LIN {X 0,Y 474.608,Z 876.179,A -85,B 0,C 180,E1 -7254.724,E2 -7254.724} C_VEL
LIN {X 0,Y 474.616,Z 876.172,A -85,B 0,C 180,E1 -7257.786,E2 -7257.786} C_VEL
LIN {X 0,Y 474.574,Z 876.184,A -85,B 0,C 180,E1 -7260.895,E2 -7260.895} C_VEL
LIN {X 0,Y 474.57,Z 876.184,A -85,B 0,C 180,E1 -7263.623,E2 -7263.623} C_VEL
LIN {X 0,Y 474.646,Z 876.303,A -85,B 0,C 180,E1 -7265.768,E2 -7265.768} C_VEL
LIN {X 0,Y 476.171,Z 885.136,A -85,B 0,C 180,E1 -7267.663,E2 -7267.663} C_VEL
LIN {X 0,Y 475.761,Z 898.657,A -85,B 0,C 180,E1 -7270.362,E2 -7270.362} C_VEL
LIN {X 0,Y 475.106,Z 915.52,A -85,B 0,C 180,E1 -7273.676,E2 -7273.676} C_VEL
LIN {X 0,Y 474.617,Z 931.729,A -85,B 0,C 180,E1 -7276.845,E2 -7276.845} C_VEL
LIN {X 0,Y 476.334,Z 945.669,A -85,B 0,C 180,E1 -7277.131,E2 -7277.131} C_VEL
LIN {X 0,Y 476.068,Z 1005.948,A -85,B 0,C 180,E1 -7278.072,E2 -7278.072} C_VEL
LIN {X 0,Y 475.814,Z 1016.704,A -85,B 0,C 180,E1 -7278.336,E2 -7278.336} C_VEL
LIN {X 0,Y 475.639,Z 1025.306,A -85,B 0,C 180,E1 -7278.656,E2 -7278.656} C_VEL
LIN {X 0,Y 475.412,Z 1032.974,A -85,B 0,C 180,E1 -7279.028,E2 -7279.028} C_VEL
LIN {X 0,Y 475.18,Z 1041.593,A -85,B 0,C 180,E1 -7279.561,E2 -7279.561} C_VEL
LIN {X 0,Y 474.915,Z 1049.857,A -85,B 0,C 180,E1 -7280.201,E2 -7280.201} C_VEL
LIN {X 0,Y 474.663,Z 1057.701,A -85,B 0,C 180,E1 -7280.949,E2 -7280.949} C_VEL
LIN {X 0,Y 474.415,Z 1064.184,A -85,B 0,C 180,E1 -7281.695,E2 -7281.695} C_VEL
LIN {X 0,Y 474.228,Z 1070.364,A -85,B 0,C 180,E1 -7282.549,E2 -7282.549} C_VEL
LIN {X 0,Y 474.034,Z 1076.736,A -85,B 0,C 180,E1 -7283.626,E2 -7283.626} C_VEL
LIN {X 0,Y 473.878,Z 1082.509,A -85,B 0,C 180,E1 -7284.895,E2 -7284.895} C_VEL
LIN {X 0,Y 473.799,Z 1085.552,A -85,B 0,C 180,E1 -7285.746,E2 -7285.746} C_VEL
LIN {X 0,Y 473.852,Z 1087.914,A -85,B 0,C 180,E1 -7286.599,E2 -7286.599} C_VEL
LIN {X 0,Y 473.745,Z 1089.693,A -85,B 0,C 180,E1 -7287.449,E2 -7287.449} C_VEL
LIN {X 0,Y 473.723,Z 1090.971,A -85,B 0,C 180,E1 -7288.3,E2 -7288.3} C_VEL
LIN {X 0,Y 473.685,Z 1091.763,A -85,B 0,C 180,E1 -7289.15,E2 -7289.15} C_VEL
LIN {X 0,Y 473.666,Z 1092.054,A -85,B 0,C 180,E1 -7290,E2 -7290} C_VEL
LIN {X 0,Y 473.685,Z 1091.749,A -85,B 0,C 180,E1 -7290.85,E2 -7290.85} C_VEL
LIN {X 0,Y 473.723,Z 1090.953,A -85,B 0,C 180,E1 -7291.7,E2 -7291.7} C_VEL
LIN {X 0,Y 473.745,Z 1089.662,A -85,B 0,C 180,E1 -7292.551,E2 -7292.551} C_VEL
LIN {X 0,Y 473.852,Z 1086.693,A -85,B 0,C 180,E1 -7293.827,E2 -7293.827} C_VEL
LIN {X 0,Y 473.878,Z 1082.413,A -85,B 0,C 180,E1 -7295.105,E2 -7295.105} C_VEL
LIN {X 0,Y 474.038,Z 1076.567,A -85,B 0,C 180,E1 -7296.38,E2 -7296.38} C_VEL
LIN {X 0,Y 474.228,Z 1070.202,A -85,B 0,C 180,E1 -7297.451,E2 -7297.451} C_VEL
LIN {X 0,Y 474.391,Z 1063.985,A -85,B 0,C 180,E1 -7298.305,E2 -7298.305} C_VEL
LIN {X 0,Y 474.656,Z 1056.411,A -85,B 0,C 180,E1 -7299.159,E2 -7299.159} C_VEL
LIN {X 0,Y 474.931,Z 1048.281,A -85,B 0,C 180,E1 -7299.906,E2 -7299.906} C_VEL
LIN {X 0,Y 475.267,Z 1038.079,A -85,B 0,C 180,E1 -7300.652,E2 -7300.652} C_VEL
LIN {X 0,Y 475.519,Z 1027.086,A -85,B 0,C 180,E1 -7301.239,E2 -7301.239} C_VEL
LIN {X 0,Y 475.754,Z 1017.515,A -85,B 0,C 180,E1 -7301.611,E2 -7301.611} C_VEL
LIN {X 0,Y 475.986,Z 1008.593,A -85,B 0,C 180,E1 -7301.849,E2 -7301.849} C_VEL
LIN {X 0,Y 476.181,Z 944.23,A -85,B 0,C 180,E1 -7302.888,E2 -7302.888} C_VEL
LIN {X 0,Y 474.612,Z 931.089,A -85,B 0,C 180,E1 -7303.172,E2 -7303.172} C_VEL
LIN {X 0,Y 475.08,Z 913.604,A -85,B 0,C 180,E1 -7306.545,E2 -7306.545} C_VEL
LIN {X 0,Y 475.627,Z 897.776,A -85,B 0,C 180,E1 -7309.643,E2 -7309.643} C_VEL
LIN {X 0,Y 476.054,Z 884.31,A -85,B 0,C 180,E1 -7312.343,E2 -7312.343} C_VEL
LIN {X 0,Y 474.644,Z 876.176,A -85,B 0,C 180,E1 -7314.144,E2 -7314.144} C_VEL
LIN {X 0,Y 474.59,Z 876.184,A -85,B 0,C 180,E1 -7317.327,E2 -7317.327} C_VEL
LIN {X 0,Y 474.547,Z 876.183,A -85,B 0,C 180,E1 -7320.234,E2 -7320.234} C_VEL
LIN {X 0,Y 474.61,Z 876.182,A -85,B 0,C 180,E1 -7323.223,E2 -7323.223} C_VEL
LIN {X 0,Y 474.564,Z 876.18,A -85,B 0,C 180,E1 -7326.326,E2 -7326.326} C_VEL
LIN {X 0,Y 474.594,Z 876.182,A -85,B 0,C 180,E1 -7329.551,E2 -7329.551} C_VEL
LIN {X 0,Y 474.562,Z 876.181,A -85,B 0,C 180,E1 -7332.94,E2 -7332.94} C_VEL
LIN {X 0,Y 474.595,Z 876.182,A -85,B 0,C 180,E1 -7335.894,E2 -7335.894} C_VEL
LIN {X 0,Y 474.578,Z 876.178,A -85,B 0,C 180,E1 -7339.048,E2 -7339.048} C_VEL
LIN {X 0,Y 474.58,Z 876.181,A -85,B 0,C 180,E1 -7341.709,E2 -7341.709} C_VEL
LIN {X 0,Y 474.607,Z 876.178,A -85,B 0,C 180,E1 -7344.724,E2 -7344.724} C_VEL
LIN {X 0,Y 474.615,Z 876.175,A -85,B 0,C 180,E1 -7347.786,E2 -7347.786} C_VEL
LIN {X 0,Y 474.573,Z 876.185,A -85,B 0,C 180,E1 -7350.896,E2 -7350.896} C_VEL
LIN {X 0,Y 474.569,Z 876.181,A -85,B 0,C 180,E1 -7353.623,E2 -7353.623} C_VEL
LIN {X 0,Y 474.594,Z 876.185,A -85,B 0,C 180,E1 -7356.653,E2 -7356.653} C_VEL
LIN {X 0,Y 474.647,Z 876.177,A -85,B 0,C 180,E1 -7359.185,E2 -7359.185} C_VEL
LIN {X 0,Y 474.67,Z 876.361,A -85,B 0,C 180,E1 -7361.496,E2 -7361.496} C_VEL
LIN {X 0,Y 475.011,Z 881.021,A -85,B 0,C 180,E1 -7362.788,E2 -7362.788} C_VEL
LIN {X 0,Y 474.637,Z 892.536,A -85,B 0,C 180,E1 -7365.859,E2 -7365.859} C_VEL
LIN {X 0,Y 474.532,Z 896.576,A -85,B 0,C 180,E1 -7366.925,E2 -7366.925} C_VEL
LIN {X 0,Y 476.468,Z 909.333,A -85,B 0,C 180,E1 -7367.193,E2 -7367.193} C_VEL
LIN {X 0,Y 475.939,Z 972.842,A -85,B 0,C 180,E1 -7368.232,E2 -7368.232} C_VEL
LIN {X 0,Y 475.768,Z 983.733,A -85,B 0,C 180,E1 -7368.551,E2 -7368.551} C_VEL
LIN {X 0,Y 475.515,Z 994.365,A -85,B 0,C 180,E1 -7369.031,E2 -7369.031} C_VEL
LIN {X 0,Y 475.301,Z 1003.198,A -85,B 0,C 180,E1 -7369.565,E2 -7369.565} C_VEL
LIN {X 0,Y 475.061,Z 1011.606,A -85,B 0,C 180,E1 -7370.205,E2 -7370.205} C_VEL
LIN {X 0,Y 474.793,Z 1019.544,A -85,B 0,C 180,E1 -7370.952,E2 -7370.952} C_VEL
LIN {X 0,Y 474.52,Z 1026.089,A -85,B 0,C 180,E1 -7371.698,E2 -7371.698} C_VEL
LIN {X 0,Y 474.314,Z 1032.298,A -85,B 0,C 180,E1 -7372.551,E2 -7372.551} C_VEL
LIN {X 0,Y 474.173,Z 1038.052,A -85,B 0,C 180,E1 -7373.515,E2 -7373.515} C_VEL
LIN {X 0,Y 474.005,Z 1042.684,A -85,B 0,C 180,E1 -7374.47,E2 -7374.47} C_VEL
LIN {X 0,Y 473.892,Z 1046.03,A -85,B 0,C 180,E1 -7375.322,E2 -7375.322} C_VEL
LIN {X 0,Y 473.894,Z 1048.738,A -85,B 0,C 180,E1 -7376.174,E2 -7376.174} C_VEL
LIN {X 0,Y 473.756,Z 1051.695,A -85,B 0,C 180,E1 -7377.45,E2 -7377.45} C_VEL
LIN {X 0,Y 473.753,Z 1052.994,A -85,B 0,C 180,E1 -7378.3,E2 -7378.3} C_VEL
LIN {X 0,Y 473.686,Z 1053.81,A -85,B 0,C 180,E1 -7379.15,E2 -7379.15} C_VEL
LIN {X 0,Y 473.667,Z 1054.103,A -85,B 0,C 180,E1 -7380,E2 -7380} C_VEL
LIN {X 0,Y 473.686,Z 1053.826,A -85,B 0,C 180,E1 -7380.851,E2 -7380.851} C_VEL
LIN {X 0,Y 473.753,Z 1053.066,A -85,B 0,C 180,E1 -7381.701,E2 -7381.701} C_VEL
LIN {X 0,Y 473.746,Z 1051.823,A -85,B 0,C 180,E1 -7382.551,E2 -7382.551} C_VEL
LIN {X 0,Y 473.889,Z 1048.918,A -85,B 0,C 180,E1 -7383.827,E2 -7383.827} C_VEL
LIN {X 0,Y 473.878,Z 1044.748,A -85,B 0,C 180,E1 -7385.106,E2 -7385.106} C_VEL
LIN {X 0,Y 474.197,Z 1039.865,A -85,B 0,C 180,E1 -7386.22,E2 -7386.22} C_VEL
LIN {X 0,Y 474.292,Z 1032.814,A -85,B 0,C 180,E1 -7387.45,E2 -7387.45} C_VEL
LIN {X 0,Y 474.473,Z 1026.718,A -85,B 0,C 180,E1 -7388.304,E2 -7388.304} C_VEL
LIN {X 0,Y 474.766,Z 1019.299,A -85,B 0,C 180,E1 -7389.157,E2 -7389.157} C_VEL
LIN {X 0,Y 475.078,Z 1011.356,A -85,B 0,C 180,E1 -7389.903,E2 -7389.903} C_VEL
LIN {X 0,Y 475.355,Z 1001.42,A -85,B 0,C 180,E1 -7390.65,E2 -7390.65} C_VEL
LIN {X 0,Y 475.61,Z 990.9,A -85,B 0,C 180,E1 -7391.238,E2 -7391.238} C_VEL
LIN {X 0,Y 475.793,Z 981.013,A -85,B 0,C 180,E1 -7391.638,E2 -7391.638} C_VEL
LIN {X 0,Y 476.004,Z 971.331,A -85,B 0,C 180,E1 -7391.903,E2 -7391.903} C_VEL
LIN {X 0,Y 476.316,Z 907.193,A -85,B 0,C 180,E1 -7392.941,E2 -7392.941} C_VEL
LIN {X 0,Y 474.447,Z 895.857,A -85,B 0,C 180,E1 -7393.198,E2 -7393.198} C_VEL
LIN {X 0,Y 474.781,Z 883.788,A -85,B 0,C 180,E1 -7396.335,E2 -7396.335} C_VEL
LIN {X 0,Y 474.736,Z 876.329,A -85,B 0,C 180,E1 -7398.305,E2 -7398.305} C_VEL
LIN {X 0,Y 474.579,Z 876.178,A -85,B 0,C 180,E1 -7401.73,E2 -7401.73} C_VEL
LIN {X 0,Y 474.586,Z 876.177,A -85,B 0,C 180,E1 -7404.497,E2 -7404.497} C_VEL
LIN {X 0,Y 474.594,Z 876.184,A -85,B 0,C 180,E1 -7407.327,E2 -7407.327} C_VEL
LIN {X 0,Y 474.551,Z 876.181,A -85,B 0,C 180,E1 -7410.235,E2 -7410.235} C_VEL
LIN {X 0,Y 474.614,Z 876.176,A -85,B 0,C 180,E1 -7413.223,E2 -7413.223} C_VEL
LIN {X 0,Y 474.571,Z 876.18,A -85,B 0,C 180,E1 -7416.326,E2 -7416.326} C_VEL
LIN {X 0,Y 474.6,Z 876.178,A -85,B 0,C 180,E1 -7419.551,E2 -7419.551} C_VEL
LIN {X 0,Y 474.568,Z 876.178,A -85,B 0,C 180,E1 -7422.94,E2 -7422.94} C_VEL
LIN {X 0,Y 474.6,Z 876.179,A -85,B 0,C 180,E1 -7425.894,E2 -7425.894} C_VEL
LIN {X 0,Y 474.582,Z 876.177,A -85,B 0,C 180,E1 -7429.048,E2 -7429.048} C_VEL
LIN {X 0,Y 474.586,Z 876.177,A -85,B 0,C 180,E1 -7431.709,E2 -7431.709} C_VEL
LIN {X 0,Y 474.613,Z 876.179,A -85,B 0,C 180,E1 -7434.725,E2 -7434.725} C_VEL
LIN {X 0,Y 474.62,Z 876.172,A -85,B 0,C 180,E1 -7437.787,E2 -7437.787} C_VEL
LIN {X 0,Y 474.574,Z 876.183,A -85,B 0,C 180,E1 -7441.04,E2 -7441.04} C_VEL
LIN {X 0,Y 473.906,Z 876.263,A -85,B 0,C 180,E1 -7441.749,E2 -7441.749} C_VEL
LIN {X 0,Y 471.064,Z 876.624,A -85,B 0,C 180,E1 -7442.899,E2 -7442.899} C_VEL
LIN {X 0,Y 468.663,Z 876.918,A -85,B 0,C 180,E1 -7443.826,E2 -7443.826} C_VEL
LIN {X 0,Y 467.633,Z 877.045,A -85,B 0,C 180,E1 -7444.542,E2 -7444.542} C_VEL
LIN {X 0,Y 467.55,Z 877.056,A -85,B 0,C 180,E1 -7444.785,E2 -7444.785} C_VEL
LIN {X 0,Y 467.555,Z 877.059,A -85,B 0,C 180,E1 -7446.995,E2 -7446.995} C_VEL
LIN {X 0,Y 467.597,Z 877.049,A -85,B 0,C 180,E1 -7449.776,E2 -7449.776} C_VEL
LIN {X 0,Y 467.58,Z 877.049,A -85,B 0,C 180,E1 -7452.506,E2 -7452.506} C_VEL
LIN {X 0,Y 467.599,Z 877.051,A -85,B 0,C 180,E1 -7455.196,E2 -7455.196} C_VEL
LIN {X 0,Y 467.64,Z 877.046,A -85,B 0,C 180,E1 -7457.854,E2 -7457.854} C_VEL
LIN {X 0,Y 467.633,Z 877.046,A -85,B 0,C 180,E1 -7461.356,E2 -7461.356} C_VEL
LIN {X 0,Y 467.704,Z 877.04,A -85,B 0,C 180,E1 -7463.962,E2 -7463.962} C_VEL
LIN {X 0,Y 467.786,Z 877.025,A -85,B 0,C 180,E1 -7467.417,E2 -7467.417} C_VEL
LIN {X 0,Y 467.852,Z 877.022,A -85,B 0,C 180,E1 -7470,E2 -7470} C_VEL
LIN {X 0,Y 467.784,Z 877.027,A -85,B 0,C 180,E1 -7472.583,E2 -7472.583} C_VEL
LIN {X 0,Y 467.704,Z 877.037,A -85,B 0,C 180,E1 -7476.038,E2 -7476.038} C_VEL
LIN {X 0,Y 467.633,Z 877.048,A -85,B 0,C 180,E1 -7478.644,E2 -7478.644} C_VEL
LIN {X 0,Y 467.644,Z 877.045,A -85,B 0,C 180,E1 -7482.348,E2 -7482.348} C_VEL
LIN {X 0,Y 467.578,Z 877.049,A -85,B 0,C 180,E1 -7485.852,E2 -7485.852} C_VEL
LIN {X 0,Y 467.578,Z 877.055,A -85,B 0,C 180,E1 -7488.748,E2 -7488.748} C_VEL
LIN {X 0,Y 467.571,Z 877.055,A -85,B 0,C 180,E1 -7491.263,E2 -7491.263} C_VEL
LIN {X 0,Y 467.536,Z 877.055,A -85,B 0,C 180,E1 -7493.946,E2 -7493.946} C_VEL
LIN {X 0,Y 467.529,Z 877.057,A -85,B 0,C 180,E1 -7496.806,E2 -7496.806} C_VEL
LIN {X 0,Y 467.514,Z 877.061,A -85,B 0,C 180,E1 -7499.741,E2 -7499.741} C_VEL
LIN {X 0,Y 467.549,Z 877.053,A -85,B 0,C 180,E1 -7502.761,E2 -7502.761} C_VEL
LIN {X 0,Y 467.542,Z 877.059,A -85,B 0,C 180,E1 -7505.891,E2 -7505.891} C_VEL
LIN {X 0,Y 467.53,Z 877.056,A -85,B 0,C 180,E1 -7509.15,E2 -7509.15} C_VEL
LIN {X 0,Y 467.553,Z 877.054,A -85,B 0,C 180,E1 -7511.406,E2 -7511.406} C_VEL
LIN {X 0,Y 467.566,Z 877.051,A -85,B 0,C 180,E1 -7515.052,E2 -7515.052} C_VEL
LIN {X 0,Y 467.553,Z 877.055,A -85,B 0,C 180,E1 -7518.727,E2 -7518.727} C_VEL
LIN {X 0,Y 467.536,Z 877.057,A -85,B 0,C 180,E1 -7521.952,E2 -7521.952} C_VEL
LIN {X 0,Y 467.553,Z 877.054,A -85,B 0,C 180,E1 -7525.166,E2 -7525.166} C_VEL
LIN {X 0,Y 467.55,Z 877.055,A -85,B 0,C 180,E1 -7528.257,E2 -7528.257} C_VEL
LIN {X 0,Y 467.528,Z 877.058,A -85,B 0,C 180,E1 -7531.247,E2 -7531.247} C_VEL
LIN {X 0,Y 467.565,Z 877.052,A -85,B 0,C 180,E1 -7534.405,E2 -7534.405} C_VEL
LIN {X 0,Y 467.555,Z 877.059,A -85,B 0,C 180,E1 -7536.994,E2 -7536.994} C_VEL
LIN {X 0,Y 467.596,Z 877.048,A -85,B 0,C 180,E1 -7539.775,E2 -7539.775} C_VEL
LIN {X 0,Y 467.579,Z 877.049,A -85,B 0,C 180,E1 -7542.505,E2 -7542.505} C_VEL
LIN {X 0,Y 467.571,Z 877.055,A -85,B 0,C 180,E1 -7545.195,E2 -7545.195} C_VEL
LIN {X 0,Y 467.638,Z 877.046,A -85,B 0,C 180,E1 -7547.854,E2 -7547.854} C_VEL
LIN {X 0,Y 467.631,Z 877.046,A -85,B 0,C 180,E1 -7551.356,E2 -7551.356} C_VEL
LIN {X 0,Y 467.702,Z 877.04,A -85,B 0,C 180,E1 -7553.962,E2 -7553.962} C_VEL
LIN {X 0,Y 467.783,Z 877.025,A -85,B 0,C 180,E1 -7557.416,E2 -7557.416} C_VEL
LIN {X 0,Y 467.85,Z 877.022,A -85,B 0,C 180,E1 -7560,E2 -7560} C_VEL
LIN {X 0,Y 467.782,Z 877.027,A -85,B 0,C 180,E1 -7562.583,E2 -7562.583} C_VEL
LIN {X 0,Y 467.701,Z 877.038,A -85,B 0,C 180,E1 -7566.038,E2 -7566.038} C_VEL
LIN {X 0,Y 467.63,Z 877.048,A -85,B 0,C 180,E1 -7568.643,E2 -7568.643} C_VEL
LIN {X 0,Y 467.64,Z 877.046,A -85,B 0,C 180,E1 -7572.348,E2 -7572.348} C_VEL
LIN {X 0,Y 467.575,Z 877.049,A -85,B 0,C 180,E1 -7575.851,E2 -7575.851} C_VEL
LIN {X 0,Y 467.574,Z 877.055,A -85,B 0,C 180,E1 -7578.747,E2 -7578.747} C_VEL
LIN {X 0,Y 467.568,Z 877.055,A -85,B 0,C 180,E1 -7581.263,E2 -7581.263} C_VEL
LIN {X 0,Y 467.532,Z 877.055,A -85,B 0,C 180,E1 -7583.945,E2 -7583.945} C_VEL
LIN {X 0,Y 467.525,Z 877.058,A -85,B 0,C 180,E1 -7586.806,E2 -7586.806} C_VEL
LIN {X 0,Y 467.51,Z 877.061,A -85,B 0,C 180,E1 -7589.741,E2 -7589.741} C_VEL
LIN {X 0,Y 467.545,Z 877.053,A -85,B 0,C 180,E1 -7592.761,E2 -7592.761} C_VEL
LIN {X 0,Y 467.538,Z 877.059,A -85,B 0,C 180,E1 -7595.891,E2 -7595.891} C_VEL
LIN {X 0,Y 467.526,Z 877.056,A -85,B 0,C 180,E1 -7599.15,E2 -7599.15} C_VEL
LIN {X 0,Y 467.549,Z 877.054,A -85,B 0,C 180,E1 -7601.406,E2 -7601.406} C_VEL
LIN {X 0,Y 467.561,Z 877.051,A -85,B 0,C 180,E1 -7605.051,E2 -7605.051} C_VEL
LIN {X 0,Y 467.549,Z 877.055,A -85,B 0,C 180,E1 -7608.727,E2 -7608.727} C_VEL
LIN {X 0,Y 467.532,Z 877.057,A -85,B 0,C 180,E1 -7611.952,E2 -7611.952} C_VEL
LIN {X 0,Y 467.548,Z 877.054,A -85,B 0,C 180,E1 -7615.166,E2 -7615.166} C_VEL
LIN {X 0,Y 467.545,Z 877.056,A -85,B 0,C 180,E1 -7618.257,E2 -7618.257} C_VEL
LIN {X 0,Y 467.523,Z 877.058,A -85,B 0,C 180,E1 -7621.247,E2 -7621.247} C_VEL
LIN {X 0,Y 467.56,Z 877.059,A -85,B 0,C 180,E1 -7624.405,E2 -7624.405} C_VEL
LIN {X 0,Y 467.611,Z 877.113,A -85,B 0,C 180,E1 -7625.587,E2 -7625.587} C_VEL
LIN {X 0,Y 469.195,Z 886.106,A -85,B 0,C 180,E1 -7627.545,E2 -7627.545} C_VEL
LIN {X 0,Y 468.755,Z 899.583,A -85,B 0,C 180,E1 -7630.285,E2 -7630.285} C_VEL
LIN {X 0,Y 468.122,Z 915.269,A -85,B 0,C 180,E1 -7633.426,E2 -7633.426} C_VEL
LIN {X 0,Y 467.562,Z 931.496,A -85,B 0,C 180,E1 -7636.646,E2 -7636.646} C_VEL
LIN {X 0,Y 469.42,Z 946.323,A -85,B 0,C 180,E1 -7636.955,E2 -7636.955} C_VEL
LIN {X 0,Y 469.069,Z 1007.527,A -85,B 0,C 180,E1 -7637.946,E2 -7637.946} C_VEL
LIN {X 0,Y 468.81,Z 1017.577,A -85,B 0,C 180,E1 -7638.214,E2 -7638.214} C_VEL
LIN {X 0,Y 468.597,Z 1027.069,A -85,B 0,C 180,E1 -7638.592,E2 -7638.592} C_VEL
LIN {X 0,Y 468.297,Z 1038,A -85,B 0,C 180,E1 -7639.187,E2 -7639.187} C_VEL
LIN {X 0,Y 467.948,Z 1048.161,A -85,B 0,C 180,E1 -7639.945,E2 -7639.945} C_VEL
LIN {X 0,Y 467.617,Z 1056.243,A -85,B 0,C 180,E1 -7640.702,E2 -7640.702} C_VEL
LIN {X 0,Y 467.424,Z 1062.068,A -85,B 0,C 180,E1 -7641.352,E2 -7641.352} C_VEL
LIN {X 0,Y 467.182,Z 1068.557,A -85,B 0,C 180,E1 -7642.219,E2 -7642.219} C_VEL
LIN {X 0,Y 467.042,Z 1073.953,A -85,B 0,C 180,E1 -7643.086,E2 -7643.086} C_VEL
LIN {X 0,Y 466.926,Z 1078.452,A -85,B 0,C 180,E1 -7643.952,E2 -7643.952} C_VEL
LIN {X 0,Y 466.815,Z 1082.195,A -85,B 0,C 180,E1 -7644.817,E2 -7644.817} C_VEL
LIN {X 0,Y 466.707,Z 1085.246,A -85,B 0,C 180,E1 -7645.682,E2 -7645.682} C_VEL
LIN {X 0,Y 466.766,Z 1087.616,A -85,B 0,C 180,E1 -7646.547,E2 -7646.547} C_VEL
LIN {X 0,Y 466.668,Z 1089.404,A -85,B 0,C 180,E1 -7647.41,E2 -7647.41} C_VEL
LIN {X 0,Y 466.63,Z 1090.686,A -85,B 0,C 180,E1 -7648.274,E2 -7648.274} C_VEL
LIN {X 0,Y 466.616,Z 1091.482,A -85,B 0,C 180,E1 -7649.137,E2 -7649.137} C_VEL
LIN {X 0,Y 466.595,Z 1091.772,A -85,B 0,C 180,E1 -7650,E2 -7650} C_VEL
LIN {X 0,Y 466.616,Z 1091.463,A -85,B 0,C 180,E1 -7650.863,E2 -7650.863} C_VEL
LIN {X 0,Y 466.63,Z 1090.657,A -85,B 0,C 180,E1 -7651.726,E2 -7651.726} C_VEL
LIN {X 0,Y 466.667,Z 1089.362,A -85,B 0,C 180,E1 -7652.589,E2 -7652.589} C_VEL
LIN {X 0,Y 466.744,Z 1086.368,A -85,B 0,C 180,E1 -7653.885,E2 -7653.885} C_VEL
LIN {X 0,Y 466.815,Z 1082.069,A -85,B 0,C 180,E1 -7655.183,E2 -7655.183} C_VEL
LIN {X 0,Y 466.94,Z 1076.869,A -85,B 0,C 180,E1 -7656.35,E2 -7656.35} C_VEL
LIN {X 0,Y 467.16,Z 1069.782,A -85,B 0,C 180,E1 -7657.564,E2 -7657.564} C_VEL
LIN {X 0,Y 467.349,Z 1063.524,A -85,B 0,C 180,E1 -7658.431,E2 -7658.431} C_VEL
LIN {X 0,Y 467.593,Z 1056.95,A -85,B 0,C 180,E1 -7659.189,E2 -7659.189} C_VEL
LIN {X 0,Y 467.862,Z 1048.981,A -85,B 0,C 180,E1 -7659.947,E2 -7659.947} C_VEL
LIN {X 0,Y 468.195,Z 1040.575,A -85,B 0,C 180,E1 -7660.596,E2 -7660.596} C_VEL
LIN {X 0,Y 468.44,Z 1029.847,A -85,B 0,C 180,E1 -7661.247,E2 -7661.247} C_VEL
LIN {X 0,Y 468.716,Z 1019.047,A -85,B 0,C 180,E1 -7661.706,E2 -7661.706} C_VEL
LIN {X 0,Y 469,Z 1008.617,A -85,B 0,C 180,E1 -7662,E2 -7662} C_VEL
LIN {X 0,Y 469.312,Z 945.308,A -85,B 0,C 180,E1 -7663.056,E2 -7663.056} C_VEL
LIN {X 0,Y 467.557,Z 930.956,A -85,B 0,C 180,E1 -7663.351,E2 -7663.351} C_VEL
LIN {X 0,Y 467.945,Z 916.235,A -85,B 0,C 180,E1 -7666.222,E2 -7666.222} C_VEL
LIN {X 0,Y 468.572,Z 899.794,A -85,B 0,C 180,E1 -7669.495,E2 -7669.495} C_VEL
LIN {X 0,Y 469.119,Z 886.391,A -85,B 0,C 180,E1 -7672.227,E2 -7672.227} C_VEL
LIN {X 0,Y 467.586,Z 877.056,A -85,B 0,C 180,E1 -7674.296,E2 -7674.296} C_VEL
LIN {X 0,Y 467.535,Z 877.06,A -85,B 0,C 180,E1 -7677.774,E2 -7677.774} C_VEL
LIN {X 0,Y 467.525,Z 877.064,A -85,B 0,C 180,E1 -7681.036,E2 -7681.036} C_VEL
LIN {X 0,Y 467.564,Z 877.057,A -85,B 0,C 180,E1 -7683.79,E2 -7683.79} C_VEL
LIN {X 0,Y 467.496,Z 877.062,A -85,B 0,C 180,E1 -7686.965,E2 -7686.965} C_VEL
LIN {X 0,Y 467.519,Z 877.062,A -85,B 0,C 180,E1 -7689.946,E2 -7689.946} C_VEL
LIN {X 0,Y 467.514,Z 877.059,A -85,B 0,C 180,E1 -7692.569,E2 -7692.569} C_VEL
LIN {X 0,Y 467.559,Z 877.053,A -85,B 0,C 180,E1 -7695.052,E2 -7695.052} C_VEL
LIN {X 0,Y 467.547,Z 877.055,A -85,B 0,C 180,E1 -7698.728,E2 -7698.728} C_VEL
LIN {X 0,Y 467.531,Z 877.062,A -85,B 0,C 180,E1 -7701.953,E2 -7701.953} C_VEL
LIN {X 0,Y 467.547,Z 877.054,A -85,B 0,C 180,E1 -7705.166,E2 -7705.166} C_VEL
LIN {X 0,Y 467.544,Z 877.06,A -85,B 0,C 180,E1 -7708.257,E2 -7708.257} C_VEL
LIN {X 0,Y 467.522,Z 877.059,A -85,B 0,C 180,E1 -7711.247,E2 -7711.247} C_VEL
LIN {X 0,Y 467.559,Z 877.058,A -85,B 0,C 180,E1 -7714.406,E2 -7714.406} C_VEL
LIN {X 0,Y 467.545,Z 877.064,A -85,B 0,C 180,E1 -7716.995,E2 -7716.995} C_VEL
LIN {X 0,Y 467.591,Z 877.053,A -85,B 0,C 180,E1 -7719.776,E2 -7719.776} C_VEL
LIN {X 0,Y 467.588,Z 877.123,A -85,B 0,C 180,E1 -7721.305,E2 -7721.305} C_VEL
LIN {X 0,Y 468.029,Z 881.408,A -85,B 0,C 180,E1 -7722.523,E2 -7722.523} C_VEL
LIN {X 0,Y 467.672,Z 891.243,A -85,B 0,C 180,E1 -7725.199,E2 -7725.199} C_VEL
LIN {X 0,Y 467.527,Z 896.94,A -85,B 0,C 180,E1 -7726.726,E2 -7726.726} C_VEL
LIN {X 0,Y 469.535,Z 909.305,A -85,B 0,C 180,E1 -7727.001,E2 -7727.001} C_VEL
LIN {X 0,Y 468.987,Z 972.192,A -85,B 0,C 180,E1 -7728.055,E2 -7728.055} C_VEL
LIN {X 0,Y 468.812,Z 982.59,A -85,B 0,C 180,E1 -7728.352,E2 -7728.352} C_VEL
LIN {X 0,Y 468.527,Z 994.306,A -85,B 0,C 180,E1 -7728.865,E2 -7728.865} C_VEL
LIN {X 0,Y 468.266,Z 1004.715,A -85,B 0,C 180,E1 -7729.515,E2 -7729.515} C_VEL
LIN {X 0,Y 468.012,Z 1012.911,A -85,B 0,C 180,E1 -7730.165,E2 -7730.165} C_VEL
LIN {X 0,Y 467.729,Z 1020.686,A -85,B 0,C 180,E1 -7730.923,E2 -7730.923} C_VEL
LIN {X 0,Y 467.38,Z 1029.614,A -85,B 0,C 180,E1 -7732.005,E2 -7732.005} C_VEL
LIN {X 0,Y 467.152,Z 1036.985,A -85,B 0,C 180,E1 -7733.182,E2 -7733.182} C_VEL
LIN {X 0,Y 467.103,Z 1040.992,A -85,B 0,C 180,E1 -7733.955,E2 -7733.955} C_VEL
LIN {X 0,Y 466.826,Z 1044.754,A -85,B 0,C 180,E1 -7734.818,E2 -7734.818} C_VEL
LIN {X 0,Y 466.829,Z 1048.999,A -85,B 0,C 180,E1 -7736.116,E2 -7736.116} C_VEL
LIN {X 0,Y 466.677,Z 1051.965,A -85,B 0,C 180,E1 -7737.411,E2 -7737.411} C_VEL
LIN {X 0,Y 466.672,Z 1053.267,A -85,B 0,C 180,E1 -7738.274,E2 -7738.274} C_VEL
LIN {X 0,Y 466.617,Z 1054.087,A -85,B 0,C 180,E1 -7739.137,E2 -7739.137} C_VEL
LIN {X 0,Y 466.596,Z 1054.387,A -85,B 0,C 180,E1 -7740,E2 -7740} C_VEL
LIN {X 0,Y 466.618,Z 1054.098,A -85,B 0,C 180,E1 -7740.863,E2 -7740.863} C_VEL
LIN {X 0,Y 466.658,Z 1053.328,A -85,B 0,C 180,E1 -7741.726,E2 -7741.726} C_VEL
LIN {X 0,Y 466.668,Z 1052.079,A -85,B 0,C 180,E1 -7742.59,E2 -7742.59} C_VEL
LIN {X 0,Y 466.821,Z 1049.157,A -85,B 0,C 180,E1 -7743.885,E2 -7743.885} C_VEL
LIN {X 0,Y 466.77,Z 1046.499,A -85,B 0,C 180,E1 -7744.751,E2 -7744.751} C_VEL
LIN {X 0,Y 467.104,Z 1041.28,A -85,B 0,C 180,E1 -7746.046,E2 -7746.046} C_VEL
LIN {X 0,Y 467.187,Z 1034.39,A -85,B 0,C 180,E1 -7747.347,E2 -7747.347} C_VEL
LIN {X 0,Y 467.45,Z 1026.839,A -85,B 0,C 180,E1 -7748.43,E2 -7748.43} C_VEL
LIN {X 0,Y 467.779,Z 1019.385,A -85,B 0,C 180,E1 -7749.295,E2 -7749.295} C_VEL
LIN {X 0,Y 468.079,Z 1011.397,A -85,B 0,C 180,E1 -7750.053,E2 -7750.053} C_VEL
LIN {X 0,Y 468.396,Z 1001.408,A -85,B 0,C 180,E1 -7750.811,E2 -7750.811} C_VEL
LIN {X 0,Y 468.651,Z 990.743,A -85,B 0,C 180,E1 -7751.407,E2 -7751.407} C_VEL
LIN {X 0,Y 468.825,Z 980.714,A -85,B 0,C 180,E1 -7751.813,E2 -7751.813} C_VEL
LIN {X 0,Y 469.032,Z 972.026,A -85,B 0,C 180,E1 -7752.055,E2 -7752.055} C_VEL
LIN {X 0,Y 469.337,Z 907.501,A -85,B 0,C 180,E1 -7753.133,E2 -7753.133} C_VEL
LIN {X 0,Y 467.443,Z 896.058,A -85,B 0,C 180,E1 -7753.404,E2 -7753.404} C_VEL
LIN {X 0,Y 467.755,Z 885.53,A -85,B 0,C 180,E1 -7756.174,E2 -7756.174} C_VEL
LIN {X 0,Y 467.835,Z 878.9,A -85,B 0,C 180,E1 -7757.937,E2 -7757.937} C_VEL
LIN {X 0,Y 467.66,Z 877.046,A -85,B 0,C 180,E1 -7758.459,E2 -7758.459} C_VEL
LIN {X 0,Y 467.568,Z 877.056,A -85,B 0,C 180,E1 -7761.264,E2 -7761.264} C_VEL
LIN {X 0,Y 467.534,Z 877.055,A -85,B 0,C 180,E1 -7763.946,E2 -7763.946} C_VEL
LIN {X 0,Y 467.526,Z 877.058,A -85,B 0,C 180,E1 -7766.806,E2 -7766.806} C_VEL
LIN {X 0,Y 467.511,Z 877.062,A -85,B 0,C 180,E1 -7769.742,E2 -7769.742} C_VEL
LIN {X 0,Y 467.573,Z 877.05,A -85,B 0,C 180,E1 -7772.76,E2 -7772.76} C_VEL
LIN {X 0,Y 467.544,Z 877.059,A -85,B 0,C 180,E1 -7775.891,E2 -7775.891} C_VEL
LIN {X 0,Y 467.53,Z 877.056,A -85,B 0,C 180,E1 -7779.151,E2 -7779.151} C_VEL
LIN {X 0,Y 467.551,Z 877.054,A -85,B 0,C 180,E1 -7781.406,E2 -7781.406} C_VEL
LIN {X 0,Y 467.564,Z 877.051,A -85,B 0,C 180,E1 -7785.052,E2 -7785.052} C_VEL
LIN {X 0,Y 467.552,Z 877.055,A -85,B 0,C 180,E1 -7788.728,E2 -7788.728} C_VEL
LIN {X 0,Y 467.538,Z 877.056,A -85,B 0,C 180,E1 -7791.953,E2 -7791.953} C_VEL
LIN {X 0,Y 467.552,Z 877.054,A -85,B 0,C 180,E1 -7795.166,E2 -7795.166} C_VEL
LIN {X 0,Y 467.549,Z 877.055,A -85,B 0,C 180,E1 -7798.257,E2 -7798.257} C_VEL
LIN {X 0,Y 467.528,Z 877.058,A -85,B 0,C 180,E1 -7801.247,E2 -7801.247} C_VEL
LIN {X 0,Y 467.565,Z 877.052,A -85,B 0,C 180,E1 -7804.406,E2 -7804.406} C_VEL
LIN {X 0,Y 467.55,Z 877.056,A -85,B 0,C 180,E1 -7804.785,E2 -7804.785} C_VEL
LIN {X 0,Y 466.89,Z 877.142,A -85,B 0,C 180,E1 -7805.503,E2 -7805.503} C_VEL
LIN {X 0,Y 464.06,Z 877.496,A -85,B 0,C 180,E1 -7806.671,E2 -7806.671} C_VEL
LIN {X 0,Y 461.657,Z 877.792,A -85,B 0,C 180,E1 -7807.612,E2 -7807.612} C_VEL
LIN {X 0,Y 460.613,Z 877.919,A -85,B 0,C 180,E1 -7808.339,E2 -7808.339} C_VEL
LIN {X 0,Y 460.521,Z 877.93,A -85,B 0,C 180,E1 -7808.585,E2 -7808.585} C_VEL
LIN {X 0,Y 460.535,Z 877.934,A -85,B 0,C 180,E1 -7811.309,E2 -7811.309} C_VEL
LIN {X 0,Y 460.591,Z 877.921,A -85,B 0,C 180,E1 -7814.059,E2 -7814.059} C_VEL
LIN {X 0,Y 460.606,Z 877.924,A -85,B 0,C 180,E1 -7817.666,E2 -7817.666} C_VEL
LIN {X 0,Y 460.588,Z 877.922,A -85,B 0,C 180,E1 -7821.223,E2 -7821.223} C_VEL
LIN {X 0,Y 460.67,Z 877.917,A -85,B 0,C 180,E1 -7823.87,E2 -7823.87} C_VEL
LIN {X 0,Y 460.733,Z 877.903,A -85,B 0,C 180,E1 -7827.377,E2 -7827.377} C_VEL
LIN {X 0,Y 460.822,Z 877.898,A -85,B 0,C 180,E1 -7830,E2 -7830} C_VEL
LIN {X 0,Y 460.731,Z 877.905,A -85,B 0,C 180,E1 -7832.623,E2 -7832.623} C_VEL
LIN {X 0,Y 460.671,Z 877.914,A -85,B 0,C 180,E1 -7836.131,E2 -7836.131} C_VEL
LIN {X 0,Y 460.588,Z 877.924,A -85,B 0,C 180,E1 -7838.777,E2 -7838.777} C_VEL
LIN {X 0,Y 460.602,Z 877.923,A -85,B 0,C 180,E1 -7842.435,E2 -7842.435} C_VEL
LIN {X 0,Y 460.531,Z 877.927,A -85,B 0,C 180,E1 -7845.965,E2 -7845.965} C_VEL
LIN {X 0,Y 460.536,Z 877.934,A -85,B 0,C 180,E1 -7848.887,E2 -7848.887} C_VEL
LIN {X 0,Y 460.516,Z 877.932,A -85,B 0,C 180,E1 -7851.486,E2 -7851.486} C_VEL
LIN {X 0,Y 460.498,Z 877.931,A -85,B 0,C 180,E1 -7854.335,E2 -7854.335} C_VEL
LIN {X 0,Y 460.489,Z 877.94,A -85,B 0,C 180,E1 -7857.249,E2 -7857.249} C_VEL
LIN {X 0,Y 460.482,Z 877.934,A -85,B 0,C 180,E1 -7860.242,E2 -7860.242} C_VEL
LIN {X 0,Y 460.502,Z 877.935,A -85,B 0,C 180,E1 -7863.327,E2 -7863.327} C_VEL
LIN {X 0,Y 460.458,Z 877.937,A -85,B 0,C 180,E1 -7866.531,E2 -7866.531} C_VEL
LIN {X 0,Y 460.495,Z 877.94,A -85,B 0,C 180,E1 -7869.867,E2 -7869.867} C_VEL
LIN {X 0,Y 460.46,Z 877.936,A -85,B 0,C 180,E1 -7872.892,E2 -7872.892} C_VEL
LIN {X 0,Y 460.504,Z 877.934,A -85,B 0,C 180,E1 -7875.832,E2 -7875.832} C_VEL
LIN {X 0,Y 460.503,Z 877.931,A -85,B 0,C 180,E1 -7878.985,E2 -7878.985} C_VEL
LIN {X 0,Y 460.482,Z 877.941,A -85,B 0,C 180,E1 -7882.374,E2 -7882.374} C_VEL
LIN {X 0,Y 460.537,Z 877.926,A -85,B 0,C 180,E1 -7885.622,E2 -7885.622} C_VEL
LIN {X 0,Y 460.508,Z 877.938,A -85,B 0,C 180,E1 -7888.742,E2 -7888.742} C_VEL
LIN {X 0,Y 460.499,Z 877.931,A -85,B 0,C 180,E1 -7891.763,E2 -7891.763} C_VEL
LIN {X 0,Y 460.513,Z 877.934,A -85,B 0,C 180,E1 -7894.702,E2 -7894.702} C_VEL
LIN {X 0,Y 460.5,Z 877.933,A -85,B 0,C 180,E1 -7897.57,E2 -7897.57} C_VEL
LIN {X 0,Y 460.525,Z 877.928,A -85,B 0,C 180,E1 -7900.382,E2 -7900.382} C_VEL
LIN {X 0,Y 460.542,Z 877.931,A -85,B 0,C 180,E1 -7903.145,E2 -7903.145} C_VEL
LIN {X 0,Y 460.53,Z 877.93,A -85,B 0,C 180,E1 -7905.867,E2 -7905.867} C_VEL
LIN {X 0,Y 460.582,Z 877.921,A -85,B 0,C 180,E1 -7908.558,E2 -7908.558} C_VEL
LIN {X 0,Y 460.625,Z 877.919,A -85,B 0,C 180,E1 -7912.107,E2 -7912.107} C_VEL
LIN {X 0,Y 460.673,Z 877.909,A -85,B 0,C 180,E1 -7914.748,E2 -7914.748} C_VEL
LIN {X 0,Y 460.715,Z 877.909,A -85,B 0,C 180,E1 -7918.251,E2 -7918.251} C_VEL
LIN {X 0,Y 460.82,Z 877.898,A -85,B 0,C 180,E1 -7920,E2 -7920} C_VEL
LIN {X 0,Y 460.729,Z 877.905,A -85,B 0,C 180,E1 -7922.623,E2 -7922.623} C_VEL
LIN {X 0,Y 460.668,Z 877.915,A -85,B 0,C 180,E1 -7926.13,E2 -7926.13} C_VEL
LIN {X 0,Y 460.585,Z 877.924,A -85,B 0,C 180,E1 -7928.777,E2 -7928.777} C_VEL
LIN {X 0,Y 460.599,Z 877.924,A -85,B 0,C 180,E1 -7932.435,E2 -7932.435} C_VEL
LIN {X 0,Y 460.527,Z 877.927,A -85,B 0,C 180,E1 -7935.964,E2 -7935.964} C_VEL
LIN {X 0,Y 460.532,Z 877.935,A -85,B 0,C 180,E1 -7938.886,E2 -7938.886} C_VEL
LIN {X 0,Y 460.512,Z 877.932,A -85,B 0,C 180,E1 -7941.485,E2 -7941.485} C_VEL
LIN {X 0,Y 460.495,Z 877.932,A -85,B 0,C 180,E1 -7944.335,E2 -7944.335} C_VEL
LIN {X 0,Y 460.485,Z 877.941,A -85,B 0,C 180,E1 -7947.249,E2 -7947.249} C_VEL
LIN {X 0,Y 460.478,Z 877.934,A -85,B 0,C 180,E1 -7950.242,E2 -7950.242} C_VEL
LIN {X 0,Y 460.498,Z 877.936,A -85,B 0,C 180,E1 -7953.327,E2 -7953.327} C_VEL
LIN {X 0,Y 460.454,Z 877.937,A -85,B 0,C 180,E1 -7956.531,E2 -7956.531} C_VEL
LIN {X 0,Y 460.491,Z 877.94,A -85,B 0,C 180,E1 -7959.866,E2 -7959.866} C_VEL
LIN {X 0,Y 460.456,Z 877.936,A -85,B 0,C 180,E1 -7962.892,E2 -7962.892} C_VEL
LIN {X 0,Y 460.499,Z 877.935,A -85,B 0,C 180,E1 -7965.832,E2 -7965.832} C_VEL
LIN {X 0,Y 460.498,Z 877.932,A -85,B 0,C 180,E1 -7968.985,E2 -7968.985} C_VEL
LIN {X 0,Y 460.477,Z 877.942,A -85,B 0,C 180,E1 -7972.374,E2 -7972.374} C_VEL
LIN {X 0,Y 460.532,Z 877.927,A -85,B 0,C 180,E1 -7975.622,E2 -7975.622} C_VEL
LIN {X 0,Y 460.503,Z 877.938,A -85,B 0,C 180,E1 -7978.742,E2 -7978.742} C_VEL
LIN {X 0,Y 460.494,Z 877.931,A -85,B 0,C 180,E1 -7981.763,E2 -7981.763} C_VEL
LIN {X 0,Y 460.58,Z 878.035,A -85,B 0,C 180,E1 -7985.429,E2 -7985.429} C_VEL
LIN {X 0,Y 462.183,Z 887.038,A -85,B 0,C 180,E1 -7987.421,E2 -7987.421} C_VEL
LIN {X 0,Y 461.758,Z 900.47,A -85,B 0,C 180,E1 -7990.205,E2 -7990.205} C_VEL
LIN {X 0,Y 461.028,Z 917.051,A -85,B 0,C 180,E1 -7993.578,E2 -7993.578} C_VEL
LIN {X 0,Y 460.533,Z 931.25,A -85,B 0,C 180,E1 -7996.438,E2 -7996.438} C_VEL
LIN {X 0,Y 462.5,Z 946.965,A -85,B 0,C 180,E1 -7996.772,E2 -7996.772} C_VEL
LIN {X 0,Y 462.085,Z 1009.013,A -85,B 0,C 180,E1 -7997.817,E2 -7997.817} C_VEL
LIN {X 0,Y 461.746,Z 1020.071,A -85,B 0,C 180,E1 -7998.142,E2 -7998.142} C_VEL
LIN {X 0,Y 461.426,Z 1031.855,A -85,B 0,C 180,E1 -7998.691,E2 -7998.691} C_VEL
LIN {X 0,Y 461.195,Z 1040.587,A -85,B 0,C 180,E1 -7999.241,E2 -7999.241} C_VEL
LIN {X 0,Y 460.882,Z 1048.938,A -85,B 0,C 180,E1 -7999.9,E2 -7999.9} C_VEL
LIN {X 0,Y 460.543,Z 1056.851,A -85,B 0,C 180,E1 -8000.669,E2 -8000.669} C_VEL
LIN {X 0,Y 460.3,Z 1063.396,A -85,B 0,C 180,E1 -8001.439,E2 -8001.439} C_VEL
LIN {X 0,Y 460.083,Z 1069.627,A -85,B 0,C 180,E1 -8002.319,E2 -8002.319} C_VEL
LIN {X 0,Y 459.896,Z 1075.713,A -85,B 0,C 180,E1 -8003.368,E2 -8003.368} C_VEL
LIN {X 0,Y 459.731,Z 1081.88,A -85,B 0,C 180,E1 -8004.737,E2 -8004.737} C_VEL
LIN {X 0,Y 459.621,Z 1084.939,A -85,B 0,C 180,E1 -8005.615,E2 -8005.615} C_VEL
LIN {X 0,Y 459.663,Z 1087.317,A -85,B 0,C 180,E1 -8006.494,E2 -8006.494} C_VEL
LIN {X 0,Y 459.593,Z 1089.115,A -85,B 0,C 180,E1 -8007.37,E2 -8007.37} C_VEL
LIN {X 0,Y 459.541,Z 1090.402,A -85,B 0,C 180,E1 -8008.247,E2 -8008.247} C_VEL
LIN {X 0,Y 459.549,Z 1091.201,A -85,B 0,C 180,E1 -8009.124,E2 -8009.124} C_VEL
LIN {X 0,Y 459.527,Z 1091.49,A -85,B 0,C 180,E1 -8010,E2 -8010} C_VEL
LIN {X 0,Y 459.549,Z 1091.177,A -85,B 0,C 180,E1 -8010.876,E2 -8010.876} C_VEL
LIN {X 0,Y 459.541,Z 1090.362,A -85,B 0,C 180,E1 -8011.753,E2 -8011.753} C_VEL
LIN {X 0,Y 459.592,Z 1089.058,A -85,B 0,C 180,E1 -8012.629,E2 -8012.629} C_VEL
LIN {X 0,Y 459.638,Z 1086.042,A -85,B 0,C 180,E1 -8013.945,E2 -8013.945} C_VEL
LIN {X 0,Y 459.672,Z 1083.292,A -85,B 0,C 180,E1 -8014.824,E2 -8014.824} C_VEL
LIN {X 0,Y 459.842,Z 1077.93,A -85,B 0,C 180,E1 -8016.141,E2 -8016.141} C_VEL
LIN {X 0,Y 460.065,Z 1070.803,A -85,B 0,C 180,E1 -8017.461,E2 -8017.461} C_VEL
LIN {X 0,Y 460.221,Z 1064.8,A -85,B 0,C 180,E1 -8018.341,E2 -8018.341} C_VEL
LIN {X 0,Y 460.526,Z 1057.488,A -85,B 0,C 180,E1 -8019.221,E2 -8019.221} C_VEL
LIN {X 0,Y 460.793,Z 1049.681,A -85,B 0,C 180,E1 -8019.991,E2 -8019.991} C_VEL
LIN {X 0,Y 461.143,Z 1041.487,A -85,B 0,C 180,E1 -8020.649,E2 -8020.649} C_VEL
LIN {X 0,Y 461.369,Z 1032.985,A -85,B 0,C 180,E1 -8021.199,E2 -8021.199} C_VEL
LIN {X 0,Y 461.601,Z 1023.092,A -85,B 0,C 180,E1 -8021.694,E2 -8021.694} C_VEL
LIN {X 0,Y 461.97,Z 1011.201,A -85,B 0,C 180,E1 -8022.102,E2 -8022.102} C_VEL
LIN {X 0,Y 462.215,Z 991.036,A -85,B 0,C 180,E1 -8022.471,E2 -8022.471} C_VEL
LIN {X 0,Y 462.334,Z 945.49,A -85,B 0,C 180,E1 -8023.247,E2 -8023.247} C_VEL
LIN {X 0,Y 460.513,Z 930.402,A -85,B 0,C 180,E1 -8023.59,E2 -8023.59} C_VEL
LIN {X 0,Y 461.04,Z 914.16,A -85,B 0,C 180,E1 -8026.836,E2 -8026.836} C_VEL
LIN {X 0,Y 461.687,Z 898.481,A -85,B 0,C 180,E1 -8030.029,E2 -8030.029} C_VEL
LIN {X 0,Y 462.138,Z 887.393,A -85,B 0,C 180,E1 -8032.345,E2 -8032.345} C_VEL
LIN {X 0,Y 460.549,Z 877.933,A -85,B 0,C 180,E1 -8034.512,E2 -8034.512} C_VEL
LIN {X 0,Y 460.507,Z 877.936,A -85,B 0,C 180,E1 -8037.729,E2 -8037.729} C_VEL
LIN {X 0,Y 460.476,Z 877.937,A -85,B 0,C 180,E1 -8040.242,E2 -8040.242} C_VEL
LIN {X 0,Y 460.513,Z 877.938,A -85,B 0,C 180,E1 -8043.326,E2 -8043.326} C_VEL
LIN {X 0,Y 460.453,Z 877.938,A -85,B 0,C 180,E1 -8046.532,E2 -8046.532} C_VEL
LIN {X 0,Y 460.471,Z 877.941,A -85,B 0,C 180,E1 -8049.869,E2 -8049.869} C_VEL
LIN {X 0,Y 460.456,Z 877.938,A -85,B 0,C 180,E1 -8052.893,E2 -8052.893} C_VEL
LIN {X 0,Y 460.492,Z 877.938,A -85,B 0,C 180,E1 -8055.833,E2 -8055.833} C_VEL
LIN {X 0,Y 460.497,Z 877.932,A -85,B 0,C 180,E1 -8058.985,E2 -8058.985} C_VEL
LIN {X 0,Y 460.476,Z 877.941,A -85,B 0,C 180,E1 -8062.375,E2 -8062.375} C_VEL
LIN {X 0,Y 460.531,Z 877.929,A -85,B 0,C 180,E1 -8065.623,E2 -8065.623} C_VEL
LIN {X 0,Y 460.502,Z 877.937,A -85,B 0,C 180,E1 -8068.742,E2 -8068.742} C_VEL
LIN {X 0,Y 460.493,Z 877.934,A -85,B 0,C 180,E1 -8071.763,E2 -8071.763} C_VEL
LIN {X 0,Y 460.499,Z 877.94,A -85,B 0,C 180,E1 -8074.702,E2 -8074.702} C_VEL
LIN {X 0,Y 460.491,Z 877.939,A -85,B 0,C 180,E1 -8077.571,E2 -8077.571} C_VEL
LIN {X 0,Y 460.526,Z 877.937,A -85,B 0,C 180,E1 -8080.805,E2 -8080.805} C_VEL
LIN {X 0,Y 460.53,Z 877.938,A -85,B 0,C 180,E1 -8081.114,E2 -8081.114} C_VEL
LIN {X 0,Y 461.053,Z 881.824,A -85,B 0,C 180,E1 -8082.25,E2 -8082.25} C_VEL
LIN {X 0,Y 460.687,Z 891.633,A -85,B 0,C 180,E1 -8084.969,E2 -8084.969} C_VEL
LIN {X 0,Y 460.543,Z 897.374,A -85,B 0,C 180,E1 -8086.521,E2 -8086.521} C_VEL
LIN {X 0,Y 462.611,Z 909.541,A -85,B 0,C 180,E1 -8086.8,E2 -8086.8} C_VEL
LIN {X 0,Y 462.023,Z 973.028,A -85,B 0,C 180,E1 -8087.9,E2 -8087.9} C_VEL
LIN {X 0,Y 461.84,Z 984.012,A -85,B 0,C 180,E1 -8088.229,E2 -8088.229} C_VEL
LIN {X 0,Y 461.572,Z 994.297,A -85,B 0,C 180,E1 -8088.695,E2 -8088.695} C_VEL
LIN {X 0,Y 461.298,Z 1004.759,A -85,B 0,C 180,E1 -8089.355,E2 -8089.355} C_VEL
LIN {X 0,Y 461.034,Z 1012.996,A -85,B 0,C 180,E1 -8090.015,E2 -8090.015} C_VEL
LIN {X 0,Y 460.72,Z 1020.807,A -85,B 0,C 180,E1 -8090.784,E2 -8090.784} C_VEL
LIN {X 0,Y 460.402,Z 1028.111,A -85,B 0,C 180,E1 -8091.662,E2 -8091.662} C_VEL
LIN {X 0,Y 460.2,Z 1035.483,A -85,B 0,C 180,E1 -8092.762,E2 -8092.762} C_VEL
LIN {X 0,Y 460.062,Z 1041.224,A -85,B 0,C 180,E1 -8093.862,E2 -8093.862} C_VEL
LIN {X 0,Y 459.774,Z 1045.002,A -85,B 0,C 180,E1 -8094.738,E2 -8094.738} C_VEL
LIN {X 0,Y 459.764,Z 1049.264,A -85,B 0,C 180,E1 -8096.056,E2 -8096.056} C_VEL
LIN {X 0,Y 459.602,Z 1052.243,A -85,B 0,C 180,E1 -8097.371,E2 -8097.371} C_VEL
LIN {X 0,Y 459.58,Z 1053.551,A -85,B 0,C 180,E1 -8098.248,E2 -8098.248} C_VEL
LIN {X 0,Y 459.551,Z 1054.373,A -85,B 0,C 180,E1 -8099.124,E2 -8099.124} C_VEL
LIN {X 0,Y 459.528,Z 1054.671,A -85,B 0,C 180,E1 -8100,E2 -8100} C_VEL
LIN {X 0,Y 459.551,Z 1054.379,A -85,B 0,C 180,E1 -8100.877,E2 -8100.877} C_VEL
LIN {X 0,Y 459.567,Z 1053.606,A -85,B 0,C 180,E1 -8101.753,E2 -8101.753} C_VEL
LIN {X 0,Y 459.594,Z 1052.345,A -85,B 0,C 180,E1 -8102.63,E2 -8102.63} C_VEL
LIN {X 0,Y 459.752,Z 1049.407,A -85,B 0,C 180,E1 -8103.945,E2 -8103.945} C_VEL
LIN {X 0,Y 459.695,Z 1046.733,A -85,B 0,C 180,E1 -8104.824,E2 -8104.824} C_VEL
LIN {X 0,Y 460.04,Z 1041.486,A -85,B 0,C 180,E1 -8106.139,E2 -8106.139} C_VEL
LIN {X 0,Y 460.145,Z 1034.551,A -85,B 0,C 180,E1 -8107.46,E2 -8107.46} C_VEL
LIN {X 0,Y 460.439,Z 1026.967,A -85,B 0,C 180,E1 -8108.559,E2 -8108.559} C_VEL
LIN {X 0,Y 460.786,Z 1019.474,A -85,B 0,C 180,E1 -8109.437,E2 -8109.437} C_VEL
LIN {X 0,Y 461.085,Z 1011.442,A -85,B 0,C 180,E1 -8110.207,E2 -8110.207} C_VEL
LIN {X 0,Y 461.434,Z 1001.379,A -85,B 0,C 180,E1 -8110.976,E2 -8110.976} C_VEL
LIN {X 0,Y 461.687,Z 990.579,A -85,B 0,C 180,E1 -8111.581,E2 -8111.581} C_VEL
LIN {X 0,Y 461.877,Z 981.231,A -85,B 0,C 180,E1 -8111.966,E2 -8111.966} C_VEL
LIN {X 0,Y 462.084,Z 971.457,A -85,B 0,C 180,E1 -8112.239,E2 -8112.239} C_VEL
LIN {X 0,Y 462.44,Z 908.39,A -85,B 0,C 180,E1 -8113.314,E2 -8113.314} C_VEL
LIN {X 0,Y 460.42,Z 896.358,A -85,B 0,C 180,E1 -8113.591,E2 -8113.591} C_VEL
LIN {X 0,Y 460.755,Z 886.013,A -85,B 0,C 180,E1 -8116.346,E2 -8116.346} C_VEL
LIN {X 0,Y 460.765,Z 879.063,A -85,B 0,C 180,E1 -8118.222,E2 -8118.222} C_VEL
LIN {X 0,Y 460.612,Z 877.925,A -85,B 0,C 180,E1 -8118.573,E2 -8118.573} C_VEL
LIN {X 0,Y 460.513,Z 877.932,A -85,B 0,C 180,E1 -8121.486,E2 -8121.486} C_VEL
LIN {X 0,Y 460.497,Z 877.931,A -85,B 0,C 180,E1 -8124.335,E2 -8124.335} C_VEL
LIN {X 0,Y 460.486,Z 877.94,A -85,B 0,C 180,E1 -8127.25,E2 -8127.25} C_VEL
LIN {X 0,Y 460.479,Z 877.934,A -85,B 0,C 180,E1 -8130.243,E2 -8130.243} C_VEL
LIN {X 0,Y 460.517,Z 877.933,A -85,B 0,C 180,E1 -8133.326,E2 -8133.326} C_VEL
LIN {X 0,Y 460.46,Z 877.937,A -85,B 0,C 180,E1 -8136.532,E2 -8136.532} C_VEL
LIN {X 0,Y 460.494,Z 877.94,A -85,B 0,C 180,E1 -8139.867,E2 -8139.867} C_VEL
LIN {X 0,Y 460.458,Z 877.936,A -85,B 0,C 180,E1 -8142.893,E2 -8142.893} C_VEL
LIN {X 0,Y 460.502,Z 877.935,A -85,B 0,C 180,E1 -8145.832,E2 -8145.832} C_VEL
LIN {X 0,Y 460.501,Z 877.932,A -85,B 0,C 180,E1 -8148.986,E2 -8148.986} C_VEL
LIN {X 0,Y 460.482,Z 877.941,A -85,B 0,C 180,E1 -8152.375,E2 -8152.375} C_VEL
LIN {X 0,Y 460.536,Z 877.926,A -85,B 0,C 180,E1 -8155.623,E2 -8155.623} C_VEL
LIN {X 0,Y 460.507,Z 877.938,A -85,B 0,C 180,E1 -8158.742,E2 -8158.742} C_VEL
LIN {X 0,Y 460.499,Z 877.931,A -85,B 0,C 180,E1 -8161.764,E2 -8161.764} C_VEL
LIN {X 0,Y 460.508,Z 877.933,A -85,B 0,C 180,E1 -8164.779,E2 -8164.779} C_VEL
LIN {X 0,Y 460.5,Z 877.933,A -85,B 0,C 180,E1 -8167.571,E2 -8167.571} C_VEL
LIN {X 0,Y 460.521,Z 877.93,A -85,B 0,C 180,E1 -8168.585,E2 -8168.585} C_VEL
LIN {X 0,Y 459.833,Z 878.02,A -85,B 0,C 180,E1 -8169.315,E2 -8169.315} C_VEL
LIN {X 0,Y 456.966,Z 878.372,A -85,B 0,C 180,E1 -8170.501,E2 -8170.501} C_VEL
LIN {X 0,Y 454.562,Z 878.676,A -85,B 0,C 180,E1 -8171.458,E2 -8171.458} C_VEL
LIN {X 0,Y 453.543,Z 878.798,A -85,B 0,C 180,E1 -8172.197,E2 -8172.197} C_VEL
LIN {X 0,Y 453.466,Z 878.807,A -85,B 0,C 180,E1 -8172.448,E2 -8172.448} C_VEL
LIN {X 0,Y 453.534,Z 878.799,A -85,B 0,C 180,E1 -8174.726,E2 -8174.726} C_VEL
LIN {X 0,Y 453.569,Z 878.802,A -85,B 0,C 180,E1 -8177.471,E2 -8177.471} C_VEL
LIN {X 0,Y 453.558,Z 878.797,A -85,B 0,C 180,E1 -8181.086,E2 -8181.086} C_VEL
LIN {X 0,Y 453.638,Z 878.793,A -85,B 0,C 180,E1 -8183.774,E2 -8183.774} C_VEL
LIN {X 0,Y 453.682,Z 878.781,A -85,B 0,C 180,E1 -8187.336,E2 -8187.336} C_VEL
LIN {X 0,Y 453.771,Z 878.776,A -85,B 0,C 180,E1 -8190,E2 -8190} C_VEL
LIN {X 0,Y 453.681,Z 878.783,A -85,B 0,C 180,E1 -8192.664,E2 -8192.664} C_VEL
LIN {X 0,Y 453.639,Z 878.792,A -85,B 0,C 180,E1 -8196.226,E2 -8196.226} C_VEL
LIN {X 0,Y 453.559,Z 878.798,A -85,B 0,C 180,E1 -8198.914,E2 -8198.914} C_VEL
LIN {X 0,Y 453.57,Z 878.801,A -85,B 0,C 180,E1 -8202.529,E2 -8202.529} C_VEL
LIN {X 0,Y 453.496,Z 878.804,A -85,B 0,C 180,E1 -8206.198,E2 -8206.198} C_VEL
LIN {X 0,Y 453.491,Z 878.811,A -85,B 0,C 180,E1 -8209.027,E2 -8209.027} C_VEL
LIN {X 0,Y 453.475,Z 878.807,A -85,B 0,C 180,E1 -8211.836,E2 -8211.836} C_VEL
LIN {X 0,Y 453.454,Z 878.811,A -85,B 0,C 180,E1 -8214.738,E2 -8214.738} C_VEL
LIN {X 0,Y 453.46,Z 878.809,A -85,B 0,C 180,E1 -8217.941,E2 -8217.941} C_VEL
LIN {X 0,Y 453.451,Z 878.81,A -85,B 0,C 180,E1 -8220.762,E2 -8220.762} C_VEL
LIN {X 0,Y 453.456,Z 878.812,A -85,B 0,C 180,E1 -8223.915,E2 -8223.915} C_VEL
LIN {X 0,Y 453.435,Z 878.813,A -85,B 0,C 180,E1 -8227.192,E2 -8227.192} C_VEL
LIN {X 0,Y 453.468,Z 878.808,A -85,B 0,C 180,E1 -8230.612,E2 -8230.612} C_VEL
LIN {X 0,Y 453.48,Z 878.808,A -85,B 0,C 180,E1 -8234.527,E2 -8234.527} C_VEL
LIN {X 0,Y 453.435,Z 878.817,A -85,B 0,C 180,E1 -8238.072,E2 -8238.072} C_VEL
LIN {X 0,Y 453.426,Z 878.815,A -85,B 0,C 180,E1 -8240.805,E2 -8240.805} C_VEL
LIN {X 0,Y 453.442,Z 878.811,A -85,B 0,C 180,E1 -8243.915,E2 -8243.915} C_VEL
LIN {X 0,Y 453.483,Z 878.81,A -85,B 0,C 180,E1 -8246.813,E2 -8246.813} C_VEL
LIN {X 0,Y 453.451,Z 878.811,A -85,B 0,C 180,E1 -8250.266,E2 -8250.266} C_VEL
LIN {X 0,Y 453.426,Z 878.815,A -85,B 0,C 180,E1 -8253.288,E2 -8253.288} C_VEL
LIN {X 0,Y 453.483,Z 878.805,A -85,B 0,C 180,E1 -8256.237,E2 -8256.237} C_VEL
LIN {X 0,Y 453.47,Z 878.814,A -85,B 0,C 180,E1 -8259.117,E2 -8259.117} C_VEL
LIN {X 0,Y 453.473,Z 878.807,A -85,B 0,C 180,E1 -8261.942,E2 -8261.942} C_VEL
LIN {X 0,Y 453.494,Z 878.804,A -85,B 0,C 180,E1 -8264.724,E2 -8264.724} C_VEL
LIN {X 0,Y 453.568,Z 878.802,A -85,B 0,C 180,E1 -8267.471,E2 -8267.471} C_VEL
LIN {X 0,Y 453.557,Z 878.797,A -85,B 0,C 180,E1 -8271.085,E2 -8271.085} C_VEL
LIN {X 0,Y 453.637,Z 878.794,A -85,B 0,C 180,E1 -8273.774,E2 -8273.774} C_VEL
LIN {X 0,Y 453.679,Z 878.781,A -85,B 0,C 180,E1 -8277.336,E2 -8277.336} C_VEL
LIN {X 0,Y 453.769,Z 878.776,A -85,B 0,C 180,E1 -8280,E2 -8280} C_VEL
LIN {X 0,Y 453.678,Z 878.783,A -85,B 0,C 180,E1 -8282.663,E2 -8282.663} C_VEL
LIN {X 0,Y 453.636,Z 878.792,A -85,B 0,C 180,E1 -8286.225,E2 -8286.225} C_VEL
LIN {X 0,Y 453.556,Z 878.799,A -85,B 0,C 180,E1 -8288.914,E2 -8288.914} C_VEL
LIN {X 0,Y 453.567,Z 878.801,A -85,B 0,C 180,E1 -8292.528,E2 -8292.528} C_VEL
LIN {X 0,Y 453.493,Z 878.805,A -85,B 0,C 180,E1 -8296.197,E2 -8296.197} C_VEL
LIN {X 0,Y 453.487,Z 878.811,A -85,B 0,C 180,E1 -8299.027,E2 -8299.027} C_VEL
LIN {X 0,Y 453.471,Z 878.807,A -85,B 0,C 180,E1 -8301.836,E2 -8301.836} C_VEL
LIN {X 0,Y 453.45,Z 878.812,A -85,B 0,C 180,E1 -8304.738,E2 -8304.738} C_VEL
LIN {X 0,Y 453.456,Z 878.81,A -85,B 0,C 180,E1 -8307.941,E2 -8307.941} C_VEL
LIN {X 0,Y 453.447,Z 878.81,A -85,B 0,C 180,E1 -8310.761,E2 -8310.761} C_VEL
LIN {X 0,Y 453.452,Z 878.813,A -85,B 0,C 180,E1 -8313.914,E2 -8313.914} C_VEL
LIN {X 0,Y 453.431,Z 878.813,A -85,B 0,C 180,E1 -8317.191,E2 -8317.191} C_VEL
LIN {X 0,Y 453.464,Z 878.808,A -85,B 0,C 180,E1 -8320.612,E2 -8320.612} C_VEL
LIN {X 0,Y 453.475,Z 878.808,A -85,B 0,C 180,E1 -8324.527,E2 -8324.527} C_VEL
LIN {X 0,Y 453.43,Z 878.818,A -85,B 0,C 180,E1 -8328.071,E2 -8328.071} C_VEL
LIN {X 0,Y 453.421,Z 878.815,A -85,B 0,C 180,E1 -8330.804,E2 -8330.804} C_VEL
LIN {X 0,Y 453.438,Z 878.812,A -85,B 0,C 180,E1 -8333.915,E2 -8333.915} C_VEL
LIN {X 0,Y 453.478,Z 878.811,A -85,B 0,C 180,E1 -8336.813,E2 -8336.813} C_VEL
LIN {X 0,Y 453.446,Z 878.812,A -85,B 0,C 180,E1 -8340.266,E2 -8340.266} C_VEL
LIN {X 0,Y 453.422,Z 878.822,A -85,B 0,C 180,E1 -8343.288,E2 -8343.288} C_VEL
LIN {X 0,Y 453.518,Z 878.941,A -85,B 0,C 180,E1 -8345.266,E2 -8345.266} C_VEL
LIN {X 0,Y 455.176,Z 887.95,A -85,B 0,C 180,E1 -8347.294,E2 -8347.294} C_VEL
LIN {X 0,Y 454.8,Z 899.131,A -85,B 0,C 180,E1 -8349.654,E2 -8349.654} C_VEL
LIN {X 0,Y 454.13,Z 914.771,A -85,B 0,C 180,E1 -8352.9,E2 -8352.9} C_VEL
LIN {X 0,Y 453.563,Z 929.399,A -85,B 0,C 180,E1 -8355.897,E2 -8355.897} C_VEL
LIN {X 0,Y 453.502,Z 931.004,A -85,B 0,C 180,E1 -8356.224,E2 -8356.224} C_VEL
LIN {X 0,Y 455.587,Z 948.327,A -85,B 0,C 180,E1 -8356.595,E2 -8356.595} C_VEL
LIN {X 0,Y 455.122,Z 1009.253,A -85,B 0,C 180,E1 -8357.656,E2 -8357.656} C_VEL
LIN {X 0,Y 454.762,Z 1020.878,A -85,B 0,C 180,E1 -8358.014,E2 -8358.014} C_VEL
LIN {X 0,Y 454.463,Z 1031.295,A -85,B 0,C 180,E1 -8358.515,E2 -8358.515} C_VEL
LIN {X 0,Y 454.197,Z 1040.083,A -85,B 0,C 180,E1 -8359.073,E2 -8359.073} C_VEL
LIN {X 0,Y 453.893,Z 1048.48,A -85,B 0,C 180,E1 -8359.743,E2 -8359.743} C_VEL
LIN {X 0,Y 453.521,Z 1056.427,A -85,B 0,C 180,E1 -8360.523,E2 -8360.523} C_VEL
LIN {X 0,Y 453.265,Z 1063.002,A -85,B 0,C 180,E1 -8361.305,E2 -8361.305} C_VEL
LIN {X 0,Y 453.015,Z 1069.259,A -85,B 0,C 180,E1 -8362.198,E2 -8362.198} C_VEL
LIN {X 0,Y 452.855,Z 1074.647,A -85,B 0,C 180,E1 -8363.129,E2 -8363.129} C_VEL
LIN {X 0,Y 452.708,Z 1079.736,A -85,B 0,C 180,E1 -8364.208,E2 -8364.208} C_VEL
LIN {X 0,Y 452.541,Z 1084.632,A -85,B 0,C 180,E1 -8365.546,E2 -8365.546} C_VEL
LIN {X 0,Y 452.56,Z 1087.017,A -85,B 0,C 180,E1 -8366.438,E2 -8366.438} C_VEL
LIN {X 0,Y 452.519,Z 1088.827,A -85,B 0,C 180,E1 -8367.329,E2 -8367.329} C_VEL
LIN {X 0,Y 452.456,Z 1090.118,A -85,B 0,C 180,E1 -8368.22,E2 -8368.22} C_VEL
LIN {X 0,Y 452.454,Z 1090.919,A -85,B 0,C 180,E1 -8369.11,E2 -8369.11} C_VEL
LIN {X 0,Y 452.46,Z 1091.207,A -85,B 0,C 180,E1 -8370,E2 -8370} C_VEL
LIN {X 0,Y 452.454,Z 1090.889,A -85,B 0,C 180,E1 -8370.89,E2 -8370.89} C_VEL
LIN {X 0,Y 452.456,Z 1090.066,A -85,B 0,C 180,E1 -8371.78,E2 -8371.78} C_VEL
LIN {X 0,Y 452.518,Z 1088.75,A -85,B 0,C 180,E1 -8372.67,E2 -8372.67} C_VEL
LIN {X 0,Y 452.536,Z 1085.717,A -85,B 0,C 180,E1 -8374.007,E2 -8374.007} C_VEL
LIN {X 0,Y 452.602,Z 1082.948,A -85,B 0,C 180,E1 -8374.899,E2 -8374.899} C_VEL
LIN {X 0,Y 452.709,Z 1079.534,A -85,B 0,C 180,E1 -8375.791,E2 -8375.791} C_VEL
LIN {X 0,Y 452.858,Z 1074.343,A -85,B 0,C 180,E1 -8376.877,E2 -8376.877} C_VEL
LIN {X 0,Y 453.008,Z 1068.934,A -85,B 0,C 180,E1 -8377.802,E2 -8377.802} C_VEL
LIN {X 0,Y 453.262,Z 1062.619,A -85,B 0,C 180,E1 -8378.695,E2 -8378.695} C_VEL
LIN {X 0,Y 453.516,Z 1055.974,A -85,B 0,C 180,E1 -8379.477,E2 -8379.477} C_VEL
LIN {X 0,Y 453.866,Z 1047.93,A -85,B 0,C 180,E1 -8380.257,E2 -8380.257} C_VEL
LIN {X 0,Y 454.206,Z 1037.893,A -85,B 0,C 180,E1 -8381.039,E2 -8381.039} C_VEL
LIN {X 0,Y 454.541,Z 1027.286,A -85,B 0,C 180,E1 -8381.652,E2 -8381.652} C_VEL
LIN {X 0,Y 454.808,Z 1017.359,A -85,B 0,C 180,E1 -8382.069,E2 -8382.069} C_VEL
LIN {X 0,Y 455.069,Z 1007.714,A -85,B 0,C 180,E1 -8382.345,E2 -8382.345} C_VEL
LIN {X 0,Y 455.432,Z 945.84,A -85,B 0,C 180,E1 -8383.44,E2 -8383.44} C_VEL
LIN {X 0,Y 453.479,Z 930.109,A -85,B 0,C 180,E1 -8383.805,E2 -8383.805} C_VEL
LIN {X 0,Y 453.988,Z 915.174,A -85,B 0,C 180,E1 -8386.85,E2 -8386.85} C_VEL
LIN {X 0,Y 454.703,Z 899.454,A -85,B 0,C 180,E1 -8390.115,E2 -8390.115} C_VEL
LIN {X 0,Y 455.164,Z 889.036,A -85,B 0,C 180,E1 -8392.334,E2 -8392.334} C_VEL
LIN {X 0,Y 453.56,Z 879.085,A -85,B 0,C 180,E1 -8394.632,E2 -8394.632} C_VEL
LIN {X 0,Y 453.515,Z 878.809,A -85,B 0,C 180,E1 -8394.734,E2 -8394.734} C_VEL
LIN {X 0,Y 453.453,Z 878.814,A -85,B 0,C 180,E1 -8397.941,E2 -8397.941} C_VEL
LIN {X 0,Y 453.444,Z 878.815,A -85,B 0,C 180,E1 -8400.762,E2 -8400.762} C_VEL
LIN {X 0,Y 453.462,Z 878.813,A -85,B 0,C 180,E1 -8403.914,E2 -8403.914} C_VEL
LIN {X 0,Y 453.429,Z 878.817,A -85,B 0,C 180,E1 -8407.192,E2 -8407.192} C_VEL
LIN {X 0,Y 453.461,Z 878.808,A -85,B 0,C 180,E1 -8410.612,E2 -8410.612} C_VEL
LIN {X 0,Y 453.476,Z 878.809,A -85,B 0,C 180,E1 -8414.528,E2 -8414.528} C_VEL
LIN {X 0,Y 453.428,Z 878.819,A -85,B 0,C 180,E1 -8418.072,E2 -8418.072} C_VEL
LIN {X 0,Y 453.42,Z 878.816,A -85,B 0,C 180,E1 -8420.805,E2 -8420.805} C_VEL
LIN {X 0,Y 453.437,Z 878.815,A -85,B 0,C 180,E1 -8423.916,E2 -8423.916} C_VEL
LIN {X 0,Y 453.477,Z 878.812,A -85,B 0,C 180,E1 -8426.813,E2 -8426.813} C_VEL
LIN {X 0,Y 453.445,Z 878.816,A -85,B 0,C 180,E1 -8430.266,E2 -8430.266} C_VEL
LIN {X 0,Y 453.421,Z 878.817,A -85,B 0,C 180,E1 -8433.289,E2 -8433.289} C_VEL
LIN {X 0,Y 453.468,Z 878.814,A -85,B 0,C 180,E1 -8436.237,E2 -8436.237} C_VEL
LIN {X 0,Y 453.464,Z 878.816,A -85,B 0,C 180,E1 -8439.117,E2 -8439.117} C_VEL
LIN {X 0,Y 453.516,Z 878.943,A -85,B 0,C 180,E1 -8440.961,E2 -8440.961} C_VEL
LIN {X 0,Y 454.075,Z 883.9,A -85,B 0,C 180,E1 -8442.434,E2 -8442.434} C_VEL
LIN {X 0,Y 453.67,Z 893.696,A -85,B 0,C 180,E1 -8445.191,E2 -8445.191} C_VEL
LIN {X 0,Y 453.543,Z 897.665,A -85,B 0,C 180,E1 -8446.292,E2 -8446.292} C_VEL
LIN {X 0,Y 455.718,Z 910.393,A -85,B 0,C 180,E1 -8446.607,E2 -8446.607} C_VEL
LIN {X 0,Y 455.074,Z 973.962,A -85,B 0,C 180,E1 -8447.74,E2 -8447.74} C_VEL
LIN {X 0,Y 454.875,Z 984.702,A -85,B 0,C 180,E1 -8448.074,E2 -8448.074} C_VEL
LIN {X 0,Y 454.566,Z 996.232,A -85,B 0,C 180,E1 -8448.631,E2 -8448.631} C_VEL
LIN {X 0,Y 454.331,Z 1004.87,A -85,B 0,C 180,E1 -8449.19,E2 -8449.19} C_VEL
LIN {X 0,Y 454.056,Z 1013.146,A -85,B 0,C 180,E1 -8449.86,E2 -8449.86} C_VEL
LIN {X 0,Y 453.784,Z 1019.962,A -85,B 0,C 180,E1 -8450.529,E2 -8450.529} C_VEL
LIN {X 0,Y 453.453,Z 1026.602,A -85,B 0,C 180,E1 -8451.309,E2 -8451.309} C_VEL
LIN {X 0,Y 453.199,Z 1032.893,A -85,B 0,C 180,E1 -8452.202,E2 -8452.202} C_VEL
LIN {X 0,Y 453.023,Z 1038.411,A -85,B 0,C 180,E1 -8453.153,E2 -8453.153} C_VEL
LIN {X 0,Y 452.878,Z 1043.403,A -85,B 0,C 180,E1 -8454.211,E2 -8454.211} C_VEL
LIN {X 0,Y 452.65,Z 1046.796,A -85,B 0,C 180,E1 -8455.102,E2 -8455.102} C_VEL
LIN {X 0,Y 452.698,Z 1049.538,A -85,B 0,C 180,E1 -8455.994,E2 -8455.994} C_VEL
LIN {X 0,Y 452.531,Z 1052.524,A -85,B 0,C 180,E1 -8457.33,E2 -8457.33} C_VEL
LIN {X 0,Y 452.492,Z 1053.836,A -85,B 0,C 180,E1 -8458.22,E2 -8458.22} C_VEL
LIN {X 0,Y 452.456,Z 1054.659,A -85,B 0,C 180,E1 -8459.11,E2 -8459.11} C_VEL
LIN {X 0,Y 452.462,Z 1054.955,A -85,B 0,C 180,E1 -8460,E2 -8460} C_VEL
LIN {X 0,Y 452.457,Z 1054.66,A -85,B 0,C 180,E1 -8460.89,E2 -8460.89} C_VEL
LIN {X 0,Y 452.48,Z 1053.878,A -85,B 0,C 180,E1 -8461.781,E2 -8461.781} C_VEL
LIN {X 0,Y 452.523,Z 1052.608,A -85,B 0,C 180,E1 -8462.671,E2 -8462.671} C_VEL
LIN {X 0,Y 452.683,Z 1049.651,A -85,B 0,C 180,E1 -8464.007,E2 -8464.007} C_VEL
LIN {X 0,Y 452.626,Z 1046.961,A -85,B 0,C 180,E1 -8464.899,E2 -8464.899} C_VEL
LIN {X 0,Y 452.971,Z 1041.69,A -85,B 0,C 180,E1 -8466.235,E2 -8466.235} C_VEL
LIN {X 0,Y 453.094,Z 1034.712,A -85,B 0,C 180,E1 -8467.577,E2 -8467.577} C_VEL
LIN {X 0,Y 453.34,Z 1028.809,A -85,B 0,C 180,E1 -8468.47,E2 -8468.47} C_VEL
LIN {X 0,Y 453.675,Z 1021.616,A -85,B 0,C 180,E1 -8469.362,E2 -8469.362} C_VEL
LIN {X 0,Y 453.99,Z 1013.958,A -85,B 0,C 180,E1 -8470.143,E2 -8470.143} C_VEL
LIN {X 0,Y 454.277,Z 1005.93,A -85,B 0,C 180,E1 -8470.812,E2 -8470.812} C_VEL
LIN {X 0,Y 454.585,Z 997.634,A -85,B 0,C 180,E1 -8471.369,E2 -8471.369} C_VEL
LIN {X 0,Y 454.748,Z 989.216,A -85,B 0,C 180,E1 -8471.817,E2 -8471.817} C_VEL
LIN {X 0,Y 454.95,Z 980.122,A -85,B 0,C 180,E1 -8472.179,E2 -8472.179} C_VEL
LIN {X 0,Y 455.189,Z 969.673,A -85,B 0,C 180,E1 -8472.456,E2 -8472.456} C_VEL
LIN {X 0,Y 455.578,Z 909.54,A -85,B 0,C 180,E1 -8473.492,E2 -8473.492} C_VEL
LIN {X 0,Y 453.379,Z 896.574,A -85,B 0,C 180,E1 -8473.806,E2 -8473.806} C_VEL
LIN {X 0,Y 453.767,Z 886.008,A -85,B 0,C 180,E1 -8476.651,E2 -8476.651} C_VEL
LIN {X 0,Y 453.642,Z 879.214,A -85,B 0,C 180,E1 -8478.518,E2 -8478.518} C_VEL
LIN {X 0,Y 453.555,Z 878.804,A -85,B 0,C 180,E1 -8478.639,E2 -8478.639} C_VEL
LIN {X 0,Y 453.472,Z 878.807,A -85,B 0,C 180,E1 -8481.837,E2 -8481.837} C_VEL
LIN {X 0,Y 453.452,Z 878.811,A -85,B 0,C 180,E1 -8484.739,E2 -8484.739} C_VEL
LIN {X 0,Y 453.457,Z 878.81,A -85,B 0,C 180,E1 -8487.941,E2 -8487.941} C_VEL
LIN {X 0,Y 453.448,Z 878.81,A -85,B 0,C 180,E1 -8490.762,E2 -8490.762} C_VEL
LIN {X 0,Y 453.466,Z 878.811,A -85,B 0,C 180,E1 -8493.914,E2 -8493.914} C_VEL
LIN {X 0,Y 453.435,Z 878.812,A -85,B 0,C 180,E1 -8497.192,E2 -8497.192} C_VEL
LIN {X 0,Y 453.466,Z 878.808,A -85,B 0,C 180,E1 -8500.613,E2 -8500.613} C_VEL
LIN {X 0,Y 453.478,Z 878.808,A -85,B 0,C 180,E1 -8504.528,E2 -8504.528} C_VEL
LIN {X 0,Y 453.433,Z 878.817,A -85,B 0,C 180,E1 -8508.072,E2 -8508.072} C_VEL
LIN {X 0,Y 453.425,Z 878.815,A -85,B 0,C 180,E1 -8510.805,E2 -8510.805} C_VEL
LIN {X 0,Y 453.443,Z 878.811,A -85,B 0,C 180,E1 -8513.916,E2 -8513.916} C_VEL
LIN {X 0,Y 453.482,Z 878.81,A -85,B 0,C 180,E1 -8516.814,E2 -8516.814} C_VEL
LIN {X 0,Y 453.45,Z 878.811,A -85,B 0,C 180,E1 -8520.267,E2 -8520.267} C_VEL
LIN {X 0,Y 453.426,Z 878.815,A -85,B 0,C 180,E1 -8523.289,E2 -8523.289} C_VEL
LIN {X 0,Y 453.483,Z 878.805,A -85,B 0,C 180,E1 -8526.238,E2 -8526.238} C_VEL
LIN {X 0,Y 453.47,Z 878.814,A -85,B 0,C 180,E1 -8529.117,E2 -8529.117} C_VEL
LIN {X 0,Y 453.474,Z 878.807,A -85,B 0,C 180,E1 -8531.943,E2 -8531.943} C_VEL
LIN {X 0,Y 453.466,Z 878.807,A -85,B 0,C 180,E1 -8532.448,E2 -8532.448} C_VEL
LIN {X 0,Y 452.817,Z 878.894,A -85,B 0,C 180,E1 -8533.189,E2 -8533.189} C_VEL
LIN {X 0,Y 449.975,Z 879.245,A -85,B 0,C 180,E1 -8534.393,E2 -8534.393} C_VEL
LIN {X 0,Y 447.566,Z 879.549,A -85,B 0,C 180,E1 -8535.364,E2 -8535.364} C_VEL
LIN {X 0,Y 446.54,Z 879.672,A -85,B 0,C 180,E1 -8536.115,E2 -8536.115} C_VEL
LIN {X 0,Y 446.461,Z 879.68,A -85,B 0,C 180,E1 -8536.369,E2 -8536.369} C_VEL
LIN {X 0,Y 446.452,Z 879.683,A -85,B 0,C 180,E1 -8539.111,E2 -8539.111} C_VEL
LIN {X 0,Y 446.594,Z 879.664,A -85,B 0,C 180,E1 -8542.496,E2 -8542.496} C_VEL
LIN {X 0,Y 446.623,Z 879.66,A -85,B 0,C 180,E1 -8544.582,E2 -8544.582} C_VEL
LIN {X 0,Y 446.657,Z 879.661,A -85,B 0,C 180,E1 -8548.197,E2 -8548.197} C_VEL
LIN {X 0,Y 446.721,Z 879.654,A -85,B 0,C 180,E1 -8550,E2 -8550} C_VEL
LIN {X 0,Y 446.632,Z 879.661,A -85,B 0,C 180,E1 -8552.706,E2 -8552.706} C_VEL
LIN {X 0,Y 446.609,Z 879.669,A -85,B 0,C 180,E1 -8556.324,E2 -8556.324} C_VEL
LIN {X 0,Y 446.509,Z 879.675,A -85,B 0,C 180,E1 -8559.056,E2 -8559.056} C_VEL
LIN {X 0,Y 446.526,Z 879.679,A -85,B 0,C 180,E1 -8562.73,E2 -8562.73} C_VEL
LIN {X 0,Y 446.443,Z 879.685,A -85,B 0,C 180,E1 -8566.461,E2 -8566.461} C_VEL
LIN {X 0,Y 446.437,Z 879.686,A -85,B 0,C 180,E1 -8569.305,E2 -8569.305} C_VEL
LIN {X 0,Y 446.411,Z 879.686,A -85,B 0,C 180,E1 -8572.2,E2 -8572.2} C_VEL
LIN {X 0,Y 446.41,Z 879.694,A -85,B 0,C 180,E1 -8575.155,E2 -8575.155} C_VEL
LIN {X 0,Y 446.42,Z 879.685,A -85,B 0,C 180,E1 -8578.183,E2 -8578.183} C_VEL
LIN {X 0,Y 446.392,Z 879.694,A -85,B 0,C 180,E1 -8581.303,E2 -8581.303} C_VEL
LIN {X 0,Y 446.415,Z 879.686,A -85,B 0,C 180,E1 -8584.525,E2 -8584.525} C_VEL
LIN {X 0,Y 446.39,Z 879.695,A -85,B 0,C 180,E1 -8587.881,E2 -8587.881} C_VEL
LIN {X 0,Y 446.398,Z 879.688,A -85,B 0,C 180,E1 -8590.912,E2 -8590.912} C_VEL
LIN {X 0,Y 446.386,Z 879.694,A -85,B 0,C 180,E1 -8593.848,E2 -8593.848} C_VEL
LIN {X 0,Y 446.387,Z 879.693,A -85,B 0,C 180,E1 -8596.406,E2 -8596.406} C_VEL
LIN {X 0,Y 446.39,Z 879.69,A -85,B 0,C 180,E1 -8599.796,E2 -8599.796} C_VEL
LIN {X 0,Y 446.393,Z 879.689,A -85,B 0,C 180,E1 -8603.253,E2 -8603.253} C_VEL
LIN {X 0,Y 446.453,Z 879.689,A -85,B 0,C 180,E1 -8606.566,E2 -8606.566} C_VEL
LIN {X 0,Y 446.417,Z 879.686,A -85,B 0,C 180,E1 -8609.983,E2 -8609.983} C_VEL
LIN {X 0,Y 446.387,Z 879.697,A -85,B 0,C 180,E1 -8612.833,E2 -8612.833} C_VEL
LIN {X 0,Y 446.422,Z 879.685,A -85,B 0,C 180,E1 -8615.937,E2 -8615.937} C_VEL
LIN {X 0,Y 446.448,Z 879.685,A -85,B 0,C 180,E1 -8618.772,E2 -8618.772} C_VEL
LIN {X 0,Y 446.422,Z 879.688,A -85,B 0,C 180,E1 -8621.647,E2 -8621.647} C_VEL
LIN {X 0,Y 446.436,Z 879.683,A -85,B 0,C 180,E1 -8624.477,E2 -8624.477} C_VEL
LIN {X 0,Y 446.519,Z 879.679,A -85,B 0,C 180,E1 -8627.384,E2 -8627.384} C_VEL
LIN {X 0,Y 446.507,Z 879.674,A -85,B 0,C 180,E1 -8630.944,E2 -8630.944} C_VEL
LIN {X 0,Y 446.607,Z 879.668,A -85,B 0,C 180,E1 -8633.675,E2 -8633.675} C_VEL
LIN {X 0,Y 446.631,Z 879.659,A -85,B 0,C 180,E1 -8637.294,E2 -8637.294} C_VEL
LIN {X 0,Y 446.719,Z 879.655,A -85,B 0,C 180,E1 -8640,E2 -8640} C_VEL
LIN {X 0,Y 446.63,Z 879.661,A -85,B 0,C 180,E1 -8642.705,E2 -8642.705} C_VEL
LIN {X 0,Y 446.606,Z 879.669,A -85,B 0,C 180,E1 -8646.324,E2 -8646.324} C_VEL
LIN {X 0,Y 446.507,Z 879.676,A -85,B 0,C 180,E1 -8649.056,E2 -8649.056} C_VEL
LIN {X 0,Y 446.523,Z 879.679,A -85,B 0,C 180,E1 -8652.729,E2 -8652.729} C_VEL
LIN {X 0,Y 446.44,Z 879.686,A -85,B 0,C 180,E1 -8656.461,E2 -8656.461} C_VEL
LIN {X 0,Y 446.434,Z 879.686,A -85,B 0,C 180,E1 -8659.304,E2 -8659.304} C_VEL
LIN {X 0,Y 446.407,Z 879.686,A -85,B 0,C 180,E1 -8662.2,E2 -8662.2} C_VEL
LIN {X 0,Y 446.406,Z 879.694,A -85,B 0,C 180,E1 -8665.155,E2 -8665.155} C_VEL
LIN {X 0,Y 446.416,Z 879.686,A -85,B 0,C 180,E1 -8668.183,E2 -8668.183} C_VEL
LIN {X 0,Y 446.388,Z 879.695,A -85,B 0,C 180,E1 -8671.302,E2 -8671.302} C_VEL
LIN {X 0,Y 446.41,Z 879.686,A -85,B 0,C 180,E1 -8674.524,E2 -8674.524} C_VEL
LIN {X 0,Y 446.385,Z 879.695,A -85,B 0,C 180,E1 -8677.881,E2 -8677.881} C_VEL
LIN {X 0,Y 446.393,Z 879.688,A -85,B 0,C 180,E1 -8680.912,E2 -8680.912} C_VEL
LIN {X 0,Y 446.382,Z 879.695,A -85,B 0,C 180,E1 -8683.848,E2 -8683.848} C_VEL
LIN {X 0,Y 446.382,Z 879.694,A -85,B 0,C 180,E1 -8686.405,E2 -8686.405} C_VEL
LIN {X 0,Y 446.386,Z 879.691,A -85,B 0,C 180,E1 -8689.795,E2 -8689.795} C_VEL
LIN {X 0,Y 446.388,Z 879.689,A -85,B 0,C 180,E1 -8693.253,E2 -8693.253} C_VEL
LIN {X 0,Y 446.448,Z 879.689,A -85,B 0,C 180,E1 -8696.566,E2 -8696.566} C_VEL
LIN {X 0,Y 446.412,Z 879.686,A -85,B 0,C 180,E1 -8699.983,E2 -8699.983} C_VEL
LIN {X 0,Y 446.381,Z 879.698,A -85,B 0,C 180,E1 -8702.833,E2 -8702.833} C_VEL
LIN {X 0,Y 446.467,Z 879.808,A -85,B 0,C 180,E1 -8705.097,E2 -8705.097} C_VEL
LIN {X 0,Y 448.246,Z 889.752,A -85,B 0,C 180,E1 -8707.363,E2 -8707.363} C_VEL
LIN {X 0,Y 447.709,Z 902.877,A -85,B 0,C 180,E1 -8710.169,E2 -8710.169} C_VEL
LIN {X 0,Y 446.914,Z 919.144,A -85,B 0,C 180,E1 -8713.589,E2 -8713.589} C_VEL
LIN {X 0,Y 446.448,Z 930.748,A -85,B 0,C 180,E1 -8716.002,E2 -8716.002} C_VEL
LIN {X 0,Y 448.681,Z 947.924,A -85,B 0,C 180,E1 -8716.385,E2 -8716.385} C_VEL
LIN {X 0,Y 448.17,Z 1009.284,A -85,B 0,C 180,E1 -8717.49,E2 -8717.49} C_VEL
LIN {X 0,Y 447.765,Z 1021.419,A -85,B 0,C 180,E1 -8717.882,E2 -8717.882} C_VEL
LIN {X 0,Y 447.412,Z 1032.522,A -85,B 0,C 180,E1 -8718.447,E2 -8718.447} C_VEL
LIN {X 0,Y 447.139,Z 1041.022,A -85,B 0,C 180,E1 -8719.013,E2 -8719.013} C_VEL
LIN {X 0,Y 446.834,Z 1049.211,A -85,B 0,C 180,E1 -8719.693,E2 -8719.693} C_VEL
LIN {X 0,Y 446.444,Z 1056.998,A -85,B 0,C 180,E1 -8720.486,E2 -8720.486} C_VEL
LIN {X 0,Y 446.068,Z 1065.974,A -85,B 0,C 180,E1 -8721.62,E2 -8721.62} C_VEL
LIN {X 0,Y 445.823,Z 1072.897,A -85,B 0,C 180,E1 -8722.755,E2 -8722.755} C_VEL
LIN {X 0,Y 445.664,Z 1077.453,A -85,B 0,C 180,E1 -8723.662,E2 -8723.662} C_VEL
LIN {X 0,Y 445.575,Z 1081.244,A -85,B 0,C 180,E1 -8724.569,E2 -8724.569} C_VEL
LIN {X 0,Y 445.441,Z 1085.539,A -85,B 0,C 180,E1 -8725.928,E2 -8725.928} C_VEL
LIN {X 0,Y 445.447,Z 1088.535,A -85,B 0,C 180,E1 -8727.287,E2 -8727.287} C_VEL
LIN {X 0,Y 445.374,Z 1089.833,A -85,B 0,C 180,E1 -8728.191,E2 -8728.191} C_VEL
LIN {X 0,Y 445.362,Z 1090.636,A -85,B 0,C 180,E1 -8729.096,E2 -8729.096} C_VEL
LIN {X 0,Y 445.367,Z 1090.923,A -85,B 0,C 180,E1 -8730,E2 -8730} C_VEL
LIN {X 0,Y 445.362,Z 1090.603,A -85,B 0,C 180,E1 -8730.904,E2 -8730.904} C_VEL
LIN {X 0,Y 445.374,Z 1089.775,A -85,B 0,C 180,E1 -8731.808,E2 -8731.808} C_VEL
LIN {X 0,Y 445.446,Z 1088.451,A -85,B 0,C 180,E1 -8732.713,E2 -8732.713} C_VEL
LIN {X 0,Y 445.441,Z 1085.407,A -85,B 0,C 180,E1 -8734.071,E2 -8734.071} C_VEL
LIN {X 0,Y 445.575,Z 1081.051,A -85,B 0,C 180,E1 -8735.43,E2 -8735.43} C_VEL
LIN {X 0,Y 445.749,Z 1075.036,A -85,B 0,C 180,E1 -8736.791,E2 -8736.791} C_VEL
LIN {X 0,Y 445.912,Z 1070.012,A -85,B 0,C 180,E1 -8737.699,E2 -8737.699} C_VEL
LIN {X 0,Y 446.131,Z 1063.953,A -85,B 0,C 180,E1 -8738.607,E2 -8738.607} C_VEL
LIN {X 0,Y 446.437,Z 1056.578,A -85,B 0,C 180,E1 -8739.514,E2 -8739.514} C_VEL
LIN {X 0,Y 446.81,Z 1048.703,A -85,B 0,C 180,E1 -8740.307,E2 -8740.307} C_VEL
LIN {X 0,Y 447.139,Z 1040.419,A -85,B 0,C 180,E1 -8740.986,E2 -8740.986} C_VEL
LIN {X 0,Y 447.465,Z 1029.93,A -85,B 0,C 180,E1 -8741.667,E2 -8741.667} C_VEL
LIN {X 0,Y 447.806,Z 1018.241,A -85,B 0,C 180,E1 -8742.203,E2 -8742.203} C_VEL
LIN {X 0,Y 448.106,Z 1008.032,A -85,B 0,C 180,E1 -8742.511,E2 -8742.511} C_VEL
LIN {X 0,Y 448.537,Z 946.526,A -85,B 0,C 180,E1 -8743.64,E2 -8743.64} C_VEL
LIN {X 0,Y 446.434,Z 929.902,A -85,B 0,C 180,E1 -8744.027,E2 -8744.027} C_VEL
LIN {X 0,Y 447.072,Z 913.752,A -85,B 0,C 180,E1 -8747.378,E2 -8747.378} C_VEL
LIN {X 0,Y 447.921,Z 897.154,A -85,B 0,C 180,E1 -8750.913,E2 -8750.913} C_VEL
LIN {X 0,Y 448.129,Z 889.362,A -85,B 0,C 180,E1 -8752.629,E2 -8752.629} C_VEL
LIN {X 0,Y 446.467,Z 879.688,A -85,B 0,C 180,E1 -8754.965,E2 -8754.965} C_VEL
LIN {X 0,Y 446.413,Z 879.691,A -85,B 0,C 180,E1 -8758.184,E2 -8758.184} C_VEL
LIN {X 0,Y 446.388,Z 879.697,A -85,B 0,C 180,E1 -8761.302,E2 -8761.302} C_VEL
LIN {X 0,Y 446.417,Z 879.689,A -85,B 0,C 180,E1 -8764.524,E2 -8764.524} C_VEL
LIN {X 0,Y 446.389,Z 879.694,A -85,B 0,C 180,E1 -8768.075,E2 -8768.075} C_VEL
LIN {X 0,Y 446.392,Z 879.693,A -85,B 0,C 180,E1 -8771.395,E2 -8771.395} C_VEL
LIN {X 0,Y 446.416,Z 879.687,A -85,B 0,C 180,E1 -8774.892,E2 -8774.892} C_VEL
LIN {X 0,Y 446.392,Z 879.691,A -85,B 0,C 180,E1 -8778.605,E2 -8778.605} C_VEL
LIN {X 0,Y 446.383,Z 879.695,A -85,B 0,C 180,E1 -8782.119,E2 -8782.119} C_VEL
LIN {X 0,Y 446.417,Z 879.687,A -85,B 0,C 180,E1 -8785.476,E2 -8785.476} C_VEL
LIN {X 0,Y 446.389,Z 879.696,A -85,B 0,C 180,E1 -8788.698,E2 -8788.698} C_VEL
LIN {X 0,Y 446.399,Z 879.69,A -85,B 0,C 180,E1 -8791.842,E2 -8791.842} C_VEL
LIN {X 0,Y 446.404,Z 879.696,A -85,B 0,C 180,E1 -8794.845,E2 -8794.845} C_VEL
LIN {X 0,Y 446.444,Z 879.69,A -85,B 0,C 180,E1 -8798.247,E2 -8798.247} C_VEL
LIN {X 0,Y 446.488,Z 879.866,A -85,B 0,C 180,E1 -8800.766,E2 -8800.766} C_VEL
LIN {X 0,Y 447.089,Z 884.399,A -85,B 0,C 180,E1 -8802.15,E2 -8802.15} C_VEL
LIN {X 0,Y 446.762,Z 892.514,A -85,B 0,C 180,E1 -8804.489,E2 -8804.489} C_VEL
LIN {X 0,Y 446.566,Z 898.042,A -85,B 0,C 180,E1 -8806.057,E2 -8806.057} C_VEL
LIN {X 0,Y 448.842,Z 911.058,A -85,B 0,C 180,E1 -8806.388,E2 -8806.388} C_VEL
LIN {X 0,Y 448.148,Z 973.81,A -85,B 0,C 180,E1 -8807.548,E2 -8807.548} C_VEL
LIN {X 0,Y 447.938,Z 984.641,A -85,B 0,C 180,E1 -8807.887,E2 -8807.887} C_VEL
LIN {X 0,Y 447.607,Z 996.294,A -85,B 0,C 180,E1 -8808.452,E2 -8808.452} C_VEL
LIN {X 0,Y 447.362,Z 1004.983,A -85,B 0,C 180,E1 -8809.019,E2 -8809.019} C_VEL
LIN {X 0,Y 447.09,Z 1013.299,A -85,B 0,C 180,E1 -8809.7,E2 -8809.7} C_VEL
LIN {X 0,Y 446.731,Z 1021.177,A -85,B 0,C 180,E1 -8810.492,E2 -8810.492} C_VEL
LIN {X 0,Y 446.357,Z 1028.532,A -85,B 0,C 180,E1 -8811.398,E2 -8811.398} C_VEL
LIN {X 0,Y 446.099,Z 1035.961,A -85,B 0,C 180,E1 -8812.532,E2 -8812.532} C_VEL
LIN {X 0,Y 445.959,Z 1041.743,A -85,B 0,C 180,E1 -8813.667,E2 -8813.667} C_VEL
LIN {X 0,Y 445.68,Z 1045.541,A -85,B 0,C 180,E1 -8814.571,E2 -8814.571} C_VEL
LIN {X 0,Y 445.631,Z 1049.826,A -85,B 0,C 180,E1 -8815.931,E2 -8815.931} C_VEL
LIN {X 0,Y 445.462,Z 1052.817,A -85,B 0,C 180,E1 -8817.288,E2 -8817.288} C_VEL
LIN {X 0,Y 445.407,Z 1054.13,A -85,B 0,C 180,E1 -8818.192,E2 -8818.192} C_VEL
LIN {X 0,Y 445.366,Z 1054.951,A -85,B 0,C 180,E1 -8819.096,E2 -8819.096} C_VEL
LIN {X 0,Y 445.368,Z 1055.243,A -85,B 0,C 180,E1 -8820,E2 -8820} C_VEL
LIN {X 0,Y 445.366,Z 1054.942,A -85,B 0,C 180,E1 -8820.905,E2 -8820.905} C_VEL
LIN {X 0,Y 445.396,Z 1054.149,A -85,B 0,C 180,E1 -8821.809,E2 -8821.809} C_VEL
LIN {X 0,Y 445.455,Z 1052.863,A -85,B 0,C 180,E1 -8822.713,E2 -8822.713} C_VEL
LIN {X 0,Y 445.595,Z 1049.886,A -85,B 0,C 180,E1 -8824.07,E2 -8824.07} C_VEL
LIN {X 0,Y 445.563,Z 1047.172,A -85,B 0,C 180,E1 -8824.977,E2 -8824.977} C_VEL
LIN {X 0,Y 445.913,Z 1041.871,A -85,B 0,C 180,E1 -8826.335,E2 -8826.335} C_VEL
LIN {X 0,Y 446.048,Z 1034.826,A -85,B 0,C 180,E1 -8827.697,E2 -8827.697} C_VEL
LIN {X 0,Y 446.316,Z 1028.879,A -85,B 0,C 180,E1 -8828.604,E2 -8828.604} C_VEL
LIN {X 0,Y 446.672,Z 1021.635,A -85,B 0,C 180,E1 -8829.51,E2 -8829.51} C_VEL
LIN {X 0,Y 446.991,Z 1013.916,A -85,B 0,C 180,E1 -8830.303,E2 -8830.303} C_VEL
LIN {X 0,Y 447.283,Z 1005.811,A -85,B 0,C 180,E1 -8830.983,E2 -8830.983} C_VEL
LIN {X 0,Y 447.591,Z 997.419,A -85,B 0,C 180,E1 -8831.549,E2 -8831.549} C_VEL
LIN {X 0,Y 447.808,Z 988.87,A -85,B 0,C 180,E1 -8832.003,E2 -8832.003} C_VEL
LIN {X 0,Y 448.059,Z 978.764,A -85,B 0,C 180,E1 -8832.398,E2 -8832.398} C_VEL
LIN {X 0,Y 448.267,Z 964.316,A -85,B 0,C 180,E1 -8832.731,E2 -8832.731} C_VEL
LIN {X 0,Y 448.617,Z 909.924,A -85,B 0,C 180,E1 -8833.685,E2 -8833.685} C_VEL
LIN {X 0,Y 446.379,Z 896.828,A -85,B 0,C 180,E1 -8834.009,E2 -8834.009} C_VEL
LIN {X 0,Y 446.769,Z 886.176,A -85,B 0,C 180,E1 -8836.919,E2 -8836.919} C_VEL
LIN {X 0,Y 446.617,Z 880.274,A -85,B 0,C 180,E1 -8838.564,E2 -8838.564} C_VEL
LIN {X 0,Y 446.507,Z 879.682,A -85,B 0,C 180,E1 -8838.789,E2 -8838.789} C_VEL
LIN {X 0,Y 446.409,Z 879.687,A -85,B 0,C 180,E1 -8842.201,E2 -8842.201} C_VEL
LIN {X 0,Y 446.408,Z 879.694,A -85,B 0,C 180,E1 -8845.156,E2 -8845.156} C_VEL
LIN {X 0,Y 446.416,Z 879.686,A -85,B 0,C 180,E1 -8848.184,E2 -8848.184} C_VEL
LIN {X 0,Y 446.392,Z 879.694,A -85,B 0,C 180,E1 -8851.303,E2 -8851.303} C_VEL
LIN {X 0,Y 446.421,Z 879.685,A -85,B 0,C 180,E1 -8854.524,E2 -8854.524} C_VEL
LIN {X 0,Y 446.396,Z 879.692,A -85,B 0,C 180,E1 -8858.076,E2 -8858.076} C_VEL
LIN {X 0,Y 446.397,Z 879.689,A -85,B 0,C 180,E1 -8861.395,E2 -8861.395} C_VEL
LIN {X 0,Y 446.42,Z 879.685,A -85,B 0,C 180,E1 -8865.109,E2 -8865.109} C_VEL
LIN {X 0,Y 446.397,Z 879.691,A -85,B 0,C 180,E1 -8868.605,E2 -8868.605} C_VEL
LIN {X 0,Y 446.389,Z 879.693,A -85,B 0,C 180,E1 -8872.119,E2 -8872.119} C_VEL
LIN {X 0,Y 446.422,Z 879.685,A -85,B 0,C 180,E1 -8875.476,E2 -8875.476} C_VEL
LIN {X 0,Y 446.394,Z 879.696,A -85,B 0,C 180,E1 -8878.698,E2 -8878.698} C_VEL
LIN {X 0,Y 446.404,Z 879.687,A -85,B 0,C 180,E1 -8881.842,E2 -8881.842} C_VEL
LIN {X 0,Y 446.415,Z 879.692,A -85,B 0,C 180,E1 -8884.845,E2 -8884.845} C_VEL
LIN {X 0,Y 446.45,Z 879.681,A -85,B 0,C 180,E1 -8888.247,E2 -8888.247} C_VEL
LIN {X 0,Y 446.422,Z 879.688,A -85,B 0,C 180,E1 -8891.648,E2 -8891.648} C_VEL
LIN {X 0,Y 446.481,Z 879.677,A -85,B 0,C 180,E1 -8894.479,E2 -8894.479} C_VEL
LIN {X 0,Y 446.461,Z 879.68,A -85,B 0,C 180,E1 -8896.369,E2 -8896.369} C_VEL
LIN {X 0,Y 445.802,Z 879.766,A -85,B 0,C 180,E1 -8897.123,E2 -8897.123} C_VEL
LIN {X 0,Y 442.937,Z 880.121,A -85,B 0,C 180,E1 -8898.346,E2 -8898.346} C_VEL
LIN {X 0,Y 440.523,Z 880.424,A -85,B 0,C 180,E1 -8899.333,E2 -8899.333} C_VEL
LIN {X 0,Y 439.509,Z 880.549,A -85,B 0,C 180,E1 -8900.097,E2 -8900.097} C_VEL
LIN {X 0,Y 439.44,Z 880.555,A -85,B 0,C 180,E1 -8900.355,E2 -8900.355} C_VEL
LIN {X 0,Y 439.562,Z 880.544,A -85,B 0,C 180,E1 -8903.574,E2 -8903.574} C_VEL
LIN {X 0,Y 439.402,Z 880.561,A -85,B 0,C 180,E1 -8905.413,E2 -8905.413} C_VEL
LIN {X 0,Y 439.626,Z 880.537,A -85,B 0,C 180,E1 -8908.168,E2 -8908.168} C_VEL
LIN {X 0,Y 439.672,Z 880.532,A -85,B 0,C 180,E1 -8910,E2 -8910} C_VEL
LIN {X 0,Y 439.586,Z 880.538,A -85,B 0,C 180,E1 -8912.749,E2 -8912.749} C_VEL
LIN {X 0,Y 439.598,Z 880.535,A -85,B 0,C 180,E1 -8915.505,E2 -8915.505} C_VEL
LIN {X 0,Y 439.484,Z 880.554,A -85,B 0,C 180,E1 -8918.275,E2 -8918.275} C_VEL
LIN {X 0,Y 439.476,Z 880.551,A -85,B 0,C 180,E1 -8921.999,E2 -8921.999} C_VEL
LIN {X 0,Y 439.382,Z 880.568,A -85,B 0,C 180,E1 -8924.829,E2 -8924.829} C_VEL
LIN {X 0,Y 439.386,Z 880.562,A -85,B 0,C 180,E1 -8927.693,E2 -8927.693} C_VEL
LIN {X 0,Y 439.372,Z 880.566,A -85,B 0,C 180,E1 -8930.604,E2 -8930.604} C_VEL
LIN {X 0,Y 439.355,Z 880.567,A -85,B 0,C 180,E1 -8933.572,E2 -8933.572} C_VEL
LIN {X 0,Y 439.359,Z 880.565,A -85,B 0,C 180,E1 -8936.609,E2 -8936.609} C_VEL
LIN {X 0,Y 439.361,Z 880.568,A -85,B 0,C 180,E1 -8939.728,E2 -8939.728} C_VEL
LIN {X 0,Y 439.345,Z 880.567,A -85,B 0,C 180,E1 -8942.949,E2 -8942.949} C_VEL
LIN {X 0,Y 439.366,Z 880.565,A -85,B 0,C 180,E1 -8946.288,E2 -8946.288} C_VEL
LIN {X 0,Y 439.363,Z 880.571,A -85,B 0,C 180,E1 -8949.78,E2 -8949.78} C_VEL
LIN {X 0,Y 439.332,Z 880.569,A -85,B 0,C 180,E1 -8952.619,E2 -8952.619} C_VEL
LIN {X 0,Y 439.377,Z 880.563,A -85,B 0,C 180,E1 -8955.267,E2 -8955.267} C_VEL
LIN {X 0,Y 439.361,Z 880.566,A -85,B 0,C 180,E1 -8958.748,E2 -8958.748} C_VEL
LIN {X 0,Y 439.354,Z 880.566,A -85,B 0,C 180,E1 -8961.612,E2 -8961.612} C_VEL
LIN {X 0,Y 439.394,Z 880.564,A -85,B 0,C 180,E1 -8964.843,E2 -8964.843} C_VEL
LIN {X 0,Y 439.356,Z 880.567,A -85,B 0,C 180,E1 -8968.138,E2 -8968.138} C_VEL
LIN {X 0,Y 439.388,Z 880.561,A -85,B 0,C 180,E1 -8971.61,E2 -8971.61} C_VEL
LIN {X 0,Y 439.357,Z 880.566,A -85,B 0,C 180,E1 -8974.412,E2 -8974.412} C_VEL
LIN {X 0,Y 439.357,Z 880.568,A -85,B 0,C 180,E1 -8977.424,E2 -8977.424} C_VEL
LIN {X 0,Y 439.39,Z 880.562,A -85,B 0,C 180,E1 -8980.683,E2 -8980.683} C_VEL
LIN {X 0,Y 439.409,Z 880.559,A -85,B 0,C 180,E1 -8984.222,E2 -8984.222} C_VEL
LIN {X 0,Y 439.487,Z 880.553,A -85,B 0,C 180,E1 -8987.286,E2 -8987.286} C_VEL
LIN {X 0,Y 439.473,Z 880.55,A -85,B 0,C 180,E1 -8990.797,E2 -8990.797} C_VEL
LIN {X 0,Y 439.56,Z 880.544,A -85,B 0,C 180,E1 -8993.573,E2 -8993.573} C_VEL
LIN {X 0,Y 439.399,Z 880.562,A -85,B 0,C 180,E1 -8995.413,E2 -8995.413} C_VEL
LIN {X 0,Y 439.624,Z 880.537,A -85,B 0,C 180,E1 -8998.167,E2 -8998.167} C_VEL
LIN {X 0,Y 439.67,Z 880.533,A -85,B 0,C 180,E1 -9000,E2 -9000} C_VEL
LIN {X 0,Y 439.584,Z 880.538,A -85,B 0,C 180,E1 -9002.749,E2 -9002.749} C_VEL
LIN {X 0,Y 439.596,Z 880.535,A -85,B 0,C 180,E1 -9005.504,E2 -9005.504} C_VEL
LIN {X 0,Y 439.481,Z 880.555,A -85,B 0,C 180,E1 -9008.275,E2 -9008.275} C_VEL
LIN {X 0,Y 439.472,Z 880.551,A -85,B 0,C 180,E1 -9011.999,E2 -9011.999} C_VEL
LIN {X 0,Y 439.383,Z 880.568,A -85,B 0,C 180,E1 -9014.828,E2 -9014.828} C_VEL
LIN {X 0,Y 439.383,Z 880.562,A -85,B 0,C 180,E1 -9017.692,E2 -9017.692} C_VEL
LIN {X 0,Y 439.368,Z 880.566,A -85,B 0,C 180,E1 -9020.604,E2 -9020.604} C_VEL
LIN {X 0,Y 439.351,Z 880.568,A -85,B 0,C 180,E1 -9023.572,E2 -9023.572} C_VEL
LIN {X 0,Y 439.355,Z 880.566,A -85,B 0,C 180,E1 -9026.608,E2 -9026.608} C_VEL
LIN {X 0,Y 439.357,Z 880.568,A -85,B 0,C 180,E1 -9029.727,E2 -9029.727} C_VEL
LIN {X 0,Y 439.341,Z 880.568,A -85,B 0,C 180,E1 -9032.948,E2 -9032.948} C_VEL
LIN {X 0,Y 439.362,Z 880.565,A -85,B 0,C 180,E1 -9036.288,E2 -9036.288} C_VEL
LIN {X 0,Y 439.359,Z 880.572,A -85,B 0,C 180,E1 -9039.78,E2 -9039.78} C_VEL
LIN {X 0,Y 439.328,Z 880.569,A -85,B 0,C 180,E1 -9042.619,E2 -9042.619} C_VEL
LIN {X 0,Y 439.372,Z 880.563,A -85,B 0,C 180,E1 -9045.267,E2 -9045.267} C_VEL
LIN {X 0,Y 439.357,Z 880.567,A -85,B 0,C 180,E1 -9048.748,E2 -9048.748} C_VEL
LIN {X 0,Y 439.349,Z 880.566,A -85,B 0,C 180,E1 -9051.612,E2 -9051.612} C_VEL
LIN {X 0,Y 439.389,Z 880.564,A -85,B 0,C 180,E1 -9054.843,E2 -9054.843} C_VEL
LIN {X 0,Y 439.352,Z 880.567,A -85,B 0,C 180,E1 -9058.137,E2 -9058.137} C_VEL
LIN {X 0,Y 439.384,Z 880.562,A -85,B 0,C 180,E1 -9061.61,E2 -9061.61} C_VEL
LIN {X 0,Y 439.41,Z 880.671,A -85,B 0,C 180,E1 -9064.922,E2 -9064.922} C_VEL
LIN {X 0,Y 441.271,Z 890.939,A -85,B 0,C 180,E1 -9067.305,E2 -9067.305} C_VEL
LIN {X 0,Y 440.587,Z 905.347,A -85,B 0,C 180,E1 -9070.428,E2 -9070.428} C_VEL
LIN {X 0,Y 439.912,Z 919.479,A -85,B 0,C 180,E1 -9073.446,E2 -9073.446} C_VEL
LIN {X 0,Y 439.453,Z 930.484,A -85,B 0,C 180,E1 -9075.775,E2 -9075.775} C_VEL
LIN {X 0,Y 441.772,Z 949.664,A -85,B 0,C 180,E1 -9076.222,E2 -9076.222} C_VEL
LIN {X 0,Y 441.204,Z 1009.12,A -85,B 0,C 180,E1 -9077.319,E2 -9077.319} C_VEL
LIN {X 0,Y 440.813,Z 1020.52,A -85,B 0,C 180,E1 -9077.687,E2 -9077.687} C_VEL
LIN {X 0,Y 440.46,Z 1031.806,A -85,B 0,C 180,E1 -9078.262,E2 -9078.262} C_VEL
LIN {X 0,Y 440.154,Z 1040.389,A -85,B 0,C 180,E1 -9078.837,E2 -9078.837} C_VEL
LIN {X 0,Y 439.819,Z 1048.642,A -85,B 0,C 180,E1 -9079.527,E2 -9079.527} C_VEL
LIN {X 0,Y 439.445,Z 1056.484,A -85,B 0,C 180,E1 -9080.333,E2 -9080.333} C_VEL
LIN {X 0,Y 439.027,Z 1065.526,A -85,B 0,C 180,E1 -9081.484,E2 -9081.484} C_VEL
LIN {X 0,Y 438.781,Z 1072.496,A -85,B 0,C 180,E1 -9082.638,E2 -9082.638} C_VEL
LIN {X 0,Y 438.591,Z 1077.08,A -85,B 0,C 180,E1 -9083.559,E2 -9083.559} C_VEL
LIN {X 0,Y 438.497,Z 1080.893,A -85,B 0,C 180,E1 -9084.481,E2 -9084.481} C_VEL
LIN {X 0,Y 438.352,Z 1085.212,A -85,B 0,C 180,E1 -9085.862,E2 -9085.862} C_VEL
LIN {X 0,Y 438.376,Z 1088.226,A -85,B 0,C 180,E1 -9087.243,E2 -9087.243} C_VEL
LIN {X 0,Y 438.295,Z 1089.537,A -85,B 0,C 180,E1 -9088.162,E2 -9088.162} C_VEL
LIN {X 0,Y 438.275,Z 1090.349,A -85,B 0,C 180,E1 -9089.081,E2 -9089.081} C_VEL
LIN {X 0,Y 438.276,Z 1090.637,A -85,B 0,C 180,E1 -9090,E2 -9090} C_VEL
LIN {X 0,Y 438.275,Z 1090.317,A -85,B 0,C 180,E1 -9090.919,E2 -9090.919} C_VEL
LIN {X 0,Y 438.295,Z 1089.491,A -85,B 0,C 180,E1 -9091.838,E2 -9091.838} C_VEL
LIN {X 0,Y 438.375,Z 1088.163,A -85,B 0,C 180,E1 -9092.757,E2 -9092.757} C_VEL
LIN {X 0,Y 438.351,Z 1085.103,A -85,B 0,C 180,E1 -9094.137,E2 -9094.137} C_VEL
LIN {X 0,Y 438.466,Z 1082.314,A -85,B 0,C 180,E1 -9095.057,E2 -9095.057} C_VEL
LIN {X 0,Y 438.525,Z 1078.868,A -85,B 0,C 180,E1 -9095.979,E2 -9095.979} C_VEL
LIN {X 0,Y 438.722,Z 1073.473,A -85,B 0,C 180,E1 -9097.131,E2 -9097.131} C_VEL
LIN {X 0,Y 438.889,Z 1068.176,A -85,B 0,C 180,E1 -9098.054,E2 -9098.054} C_VEL
LIN {X 0,Y 439.191,Z 1061.801,A -85,B 0,C 180,E1 -9098.976,E2 -9098.976} C_VEL
LIN {X 0,Y 439.507,Z 1055.09,A -85,B 0,C 180,E1 -9099.782,E2 -9099.782} C_VEL
LIN {X 0,Y 439.838,Z 1046.991,A -85,B 0,C 180,E1 -9100.588,E2 -9100.588} C_VEL
LIN {X 0,Y 440.26,Z 1036.898,A -85,B 0,C 180,E1 -9101.393,E2 -9101.393} C_VEL
LIN {X 0,Y 440.604,Z 1026.165,A -85,B 0,C 180,E1 -9102.026,E2 -9102.026} C_VEL
LIN {X 0,Y 440.92,Z 1016.164,A -85,B 0,C 180,E1 -9102.455,E2 -9102.455} C_VEL
LIN {X 0,Y 441.234,Z 1006.397,A -85,B 0,C 180,E1 -9102.739,E2 -9102.739} C_VEL
LIN {X 0,Y 441.721,Z 948.033,A -85,B 0,C 180,E1 -9103.836,E2 -9103.836} C_VEL
LIN {X 0,Y 439.45,Z 929.413,A -85,B 0,C 180,E1 -9104.305,E2 -9104.305} C_VEL
LIN {X 0,Y 440.073,Z 913.618,A -85,B 0,C 180,E1 -9107.664,E2 -9107.664} C_VEL
LIN {X 0,Y 440.957,Z 898.221,A -85,B 0,C 180,E1 -9111.015,E2 -9111.015} C_VEL
LIN {X 0,Y 441.24,Z 891.537,A -85,B 0,C 180,E1 -9112.51,E2 -9112.51} C_VEL
LIN {X 0,Y 439.721,Z 882.086,A -85,B 0,C 180,E1 -9114.806,E2 -9114.806} C_VEL
LIN {X 0,Y 439.389,Z 880.569,A -85,B 0,C 180,E1 -9115.205,E2 -9115.205} C_VEL
LIN {X 0,Y 439.374,Z 880.57,A -85,B 0,C 180,E1 -9118.676,E2 -9118.676} C_VEL
LIN {X 0,Y 439.348,Z 880.571,A -85,B 0,C 180,E1 -9122.026,E2 -9122.026} C_VEL
LIN {X 0,Y 439.383,Z 880.569,A -85,B 0,C 180,E1 -9125.339,E2 -9125.339} C_VEL
LIN {X 0,Y 439.344,Z 880.569,A -85,B 0,C 180,E1 -9128.599,E2 -9128.599} C_VEL
LIN {X 0,Y 439.342,Z 880.572,A -85,B 0,C 180,E1 -9132.211,E2 -9132.211} C_VEL
LIN {X 0,Y 439.369,Z 880.566,A -85,B 0,C 180,E1 -9135.267,E2 -9135.267} C_VEL
LIN {X 0,Y 439.355,Z 880.567,A -85,B 0,C 180,E1 -9138.748,E2 -9138.748} C_VEL
LIN {X 0,Y 439.348,Z 880.57,A -85,B 0,C 180,E1 -9141.612,E2 -9141.612} C_VEL
LIN {X 0,Y 439.388,Z 880.564,A -85,B 0,C 180,E1 -9144.843,E2 -9144.843} C_VEL
LIN {X 0,Y 439.351,Z 880.571,A -85,B 0,C 180,E1 -9148.138,E2 -9148.138} C_VEL
LIN {X 0,Y 439.383,Z 880.564,A -85,B 0,C 180,E1 -9151.61,E2 -9151.61} C_VEL
LIN {X 0,Y 439.348,Z 880.573,A -85,B 0,C 180,E1 -9154.412,E2 -9154.412} C_VEL
LIN {X 0,Y 439.349,Z 880.575,A -85,B 0,C 180,E1 -9157.424,E2 -9157.424} C_VEL
LIN {X 0,Y 439.437,Z 880.728,A -85,B 0,C 180,E1 -9160.532,E2 -9160.532} C_VEL
LIN {X 0,Y 440.085,Z 884.936,A -85,B 0,C 180,E1 -9161.856,E2 -9161.856} C_VEL
LIN {X 0,Y 439.933,Z 891.569,A -85,B 0,C 180,E1 -9163.822,E2 -9163.822} C_VEL
LIN {X 0,Y 439.594,Z 898.379,A -85,B 0,C 180,E1 -9165.788,E2 -9165.788} C_VEL
LIN {X 0,Y 441.944,Z 911.339,A -85,B 0,C 180,E1 -9166.153,E2 -9166.153} C_VEL
LIN {X 0,Y 441.233,Z 974.224,A -85,B 0,C 180,E1 -9167.349,E2 -9167.349} C_VEL
LIN {X 0,Y 441.01,Z 984.985,A -85,B 0,C 180,E1 -9167.694,E2 -9167.694} C_VEL
LIN {X 0,Y 440.666,Z 996.617,A -85,B 0,C 180,E1 -9168.268,E2 -9168.268} C_VEL
LIN {X 0,Y 440.404,Z 1005.275,A -85,B 0,C 180,E1 -9168.844,E2 -9168.844} C_VEL
LIN {X 0,Y 440.118,Z 1013.571,A -85,B 0,C 180,E1 -9169.535,E2 -9169.535} C_VEL
LIN {X 0,Y 439.736,Z 1021.439,A -85,B 0,C 180,E1 -9170.34,E2 -9170.34} C_VEL
LIN {X 0,Y 439.34,Z 1028.79,A -85,B 0,C 180,E1 -9171.259,E2 -9171.259} C_VEL
LIN {X 0,Y 439.052,Z 1036.22,A -85,B 0,C 180,E1 -9172.412,E2 -9172.412} C_VEL
LIN {X 0,Y 438.915,Z 1042.01,A -85,B 0,C 180,E1 -9173.565,E2 -9173.565} C_VEL
LIN {X 0,Y 438.638,Z 1045.818,A -85,B 0,C 180,E1 -9174.484,E2 -9174.484} C_VEL
LIN {X 0,Y 438.488,Z 1048.89,A -85,B 0,C 180,E1 -9175.404,E2 -9175.404} C_VEL
LIN {X 0,Y 438.535,Z 1051.279,A -85,B 0,C 180,E1 -9176.325,E2 -9176.325} C_VEL
LIN {X 0,Y 438.396,Z 1053.113,A -85,B 0,C 180,E1 -9177.244,E2 -9177.244} C_VEL
LIN {X 0,Y 438.326,Z 1054.425,A -85,B 0,C 180,E1 -9178.163,E2 -9178.163} C_VEL
LIN {X 0,Y 438.278,Z 1055.243,A -85,B 0,C 180,E1 -9179.082,E2 -9179.082} C_VEL
LIN {X 0,Y 438.278,Z 1055.531,A -85,B 0,C 180,E1 -9180,E2 -9180} C_VEL
LIN {X 0,Y 438.278,Z 1055.221,A -85,B 0,C 180,E1 -9180.919,E2 -9180.919} C_VEL
LIN {X 0,Y 438.316,Z 1054.416,A -85,B 0,C 180,E1 -9181.838,E2 -9181.838} C_VEL
LIN {X 0,Y 438.389,Z 1053.116,A -85,B 0,C 180,E1 -9182.757,E2 -9182.757} C_VEL
LIN {X 0,Y 438.511,Z 1050.114,A -85,B 0,C 180,E1 -9184.136,E2 -9184.136} C_VEL
LIN {X 0,Y 438.504,Z 1047.378,A -85,B 0,C 180,E1 -9185.058,E2 -9185.058} C_VEL
LIN {X 0,Y 438.858,Z 1042.039,A -85,B 0,C 180,E1 -9186.437,E2 -9186.437} C_VEL
LIN {X 0,Y 439.023,Z 1034.933,A -85,B 0,C 180,E1 -9187.821,E2 -9187.821} C_VEL
LIN {X 0,Y 439.311,Z 1028.943,A -85,B 0,C 180,E1 -9188.742,E2 -9188.742} C_VEL
LIN {X 0,Y 439.663,Z 1021.649,A -85,B 0,C 180,E1 -9189.663,E2 -9189.663} C_VEL
LIN {X 0,Y 440.001,Z 1013.868,A -85,B 0,C 180,E1 -9190.469,E2 -9190.469} C_VEL
LIN {X 0,Y 440.304,Z 1005.691,A -85,B 0,C 180,E1 -9191.16,E2 -9191.16} C_VEL
LIN {X 0,Y 440.62,Z 997.206,A -85,B 0,C 180,E1 -9191.734,E2 -9191.734} C_VEL
LIN {X 0,Y 440.903,Z 987.337,A -85,B 0,C 180,E1 -9192.252,E2 -9192.252} C_VEL
LIN {X 0,Y 441.171,Z 975.259,A -85,B 0,C 180,E1 -9192.682,E2 -9192.682} C_VEL
LIN {X 0,Y 441.437,Z 953.202,A -85,B 0,C 180,E1 -9193.108,E2 -9193.108} C_VEL
LIN {X 0,Y 441.703,Z 910.775,A -85,B 0,C 180,E1 -9193.873,E2 -9193.873} C_VEL
LIN {X 0,Y 439.365,Z 897.097,A -85,B 0,C 180,E1 -9194.215,E2 -9194.215} C_VEL
LIN {X 0,Y 439.775,Z 886.331,A -85,B 0,C 180,E1 -9197.197,E2 -9197.197} C_VEL
LIN {X 0,Y 439.47,Z 880.559,A -85,B 0,C 180,E1 -9198.836,E2 -9198.836} C_VEL
LIN {X 0,Y 439.384,Z 880.562,A -85,B 0,C 180,E1 -9201.918,E2 -9201.918} C_VEL
LIN {X 0,Y 439.377,Z 880.563,A -85,B 0,C 180,E1 -9204.575,E2 -9204.575} C_VEL
LIN {X 0,Y 439.331,Z 880.572,A -85,B 0,C 180,E1 -9207.641,E2 -9207.641} C_VEL
LIN {X 0,Y 439.344,Z 880.567,A -85,B 0,C 180,E1 -9210.79,E2 -9210.79} C_VEL
LIN {X 0,Y 439.359,Z 880.567,A -85,B 0,C 180,E1 -9214.047,E2 -9214.047} C_VEL
LIN {X 0,Y 439.338,Z 880.567,A -85,B 0,C 180,E1 -9216.885,E2 -9216.885} C_VEL
LIN {X 0,Y 439.347,Z 880.574,A -85,B 0,C 180,E1 -9219.841,E2 -9219.841} C_VEL
LIN {X 0,Y 439.33,Z 880.569,A -85,B 0,C 180,E1 -9222.62,E2 -9222.62} C_VEL
LIN {X 0,Y 439.375,Z 880.563,A -85,B 0,C 180,E1 -9225.267,E2 -9225.267} C_VEL
LIN {X 0,Y 439.36,Z 880.567,A -85,B 0,C 180,E1 -9228.748,E2 -9228.748} C_VEL
LIN {X 0,Y 439.353,Z 880.566,A -85,B 0,C 180,E1 -9231.612,E2 -9231.612} C_VEL
LIN {X 0,Y 439.394,Z 880.564,A -85,B 0,C 180,E1 -9234.844,E2 -9234.844} C_VEL
LIN {X 0,Y 439.356,Z 880.567,A -85,B 0,C 180,E1 -9238.138,E2 -9238.138} C_VEL
LIN {X 0,Y 439.388,Z 880.562,A -85,B 0,C 180,E1 -9241.61,E2 -9241.61} C_VEL
LIN {X 0,Y 439.357,Z 880.566,A -85,B 0,C 180,E1 -9244.412,E2 -9244.412} C_VEL
LIN {X 0,Y 439.357,Z 880.568,A -85,B 0,C 180,E1 -9247.424,E2 -9247.424} C_VEL
LIN {X 0,Y 439.39,Z 880.562,A -85,B 0,C 180,E1 -9250.684,E2 -9250.684} C_VEL
LIN {X 0,Y 439.449,Z 880.554,A -85,B 0,C 180,E1 -9254.224,E2 -9254.224} C_VEL
LIN {X 0,Y 439.475,Z 880.553,A -85,B 0,C 180,E1 -9258.001,E2 -9258.001} C_VEL
LIN {X 0,Y 439.44,Z 880.555,A -85,B 0,C 180,E1 -9260.355,E2 -9260.355} C_VEL
LIN {X 0,Y 438.85,Z 880.63,A -85,B 0,C 180,E1 -9261.12,E2 -9261.12} C_VEL
LIN {X 0,Y 436.164,Z 880.966,A -85,B 0,C 180,E1 -9262.365,E2 -9262.365} C_VEL
LIN {X 0,Y 432.961,Z 881.368,A -85,B 0,C 180,E1 -9263.883,E2 -9263.883} C_VEL
LIN {X 0,Y 432.554,Z 881.414,A -85,B 0,C 180,E1 -9264.406,E2 -9264.406} C_VEL
LIN {X 0,Y 432.595,Z 881.413,A -85,B 0,C 180,E1 -9268.138,E2 -9268.138} C_VEL
LIN {X 0,Y 432.624,Z 881.41,A -85,B 0,C 180,E1 -9270,E2 -9270} C_VEL
LIN {X 0,Y 432.541,Z 881.415,A -85,B 0,C 180,E1 -9272.794,E2 -9272.794} C_VEL
LIN {X 0,Y 432.554,Z 881.413,A -85,B 0,C 180,E1 -9275.595,E2 -9275.595} C_VEL
LIN {X 0,Y 432.45,Z 881.432,A -85,B 0,C 180,E1 -9278.411,E2 -9278.411} C_VEL
LIN {X 0,Y 432.455,Z 881.427,A -85,B 0,C 180,E1 -9282.197,E2 -9282.197} C_VEL
LIN {X 0,Y 432.365,Z 881.436,A -85,B 0,C 180,E1 -9286.042,E2 -9286.042} C_VEL
LIN {X 0,Y 432.352,Z 881.439,A -85,B 0,C 180,E1 -9289.47,E2 -9289.47} C_VEL
LIN {X 0,Y 432.343,Z 881.439,A -85,B 0,C 180,E1 -9292.092,E2 -9292.092} C_VEL
LIN {X 0,Y 432.316,Z 881.447,A -85,B 0,C 180,E1 -9295.004,E2 -9295.004} C_VEL
LIN {X 0,Y 432.316,Z 881.442,A -85,B 0,C 180,E1 -9298.128,E2 -9298.128} C_VEL
LIN {X 0,Y 432.303,Z 881.45,A -85,B 0,C 180,E1 -9301.348,E2 -9301.348} C_VEL
LIN {X 0,Y 432.325,Z 881.441,A -85,B 0,C 180,E1 -9304.679,E2 -9304.679} C_VEL
LIN {X 0,Y 432.321,Z 881.444,A -85,B 0,C 180,E1 -9308.152,E2 -9308.152} C_VEL
LIN {X 0,Y 432.304,Z 881.449,A -85,B 0,C 180,E1 -9311.801,E2 -9311.801} C_VEL
LIN {X 0,Y 432.335,Z 881.443,A -85,B 0,C 180,E1 -9314.348,E2 -9314.348} C_VEL
LIN {X 0,Y 432.305,Z 881.444,A -85,B 0,C 180,E1 -9317.018,E2 -9317.018} C_VEL
LIN {X 0,Y 432.291,Z 881.447,A -85,B 0,C 180,E1 -9319.828,E2 -9319.828} C_VEL
LIN {X 0,Y 432.297,Z 881.446,A -85,B 0,C 180,E1 -9323.02,E2 -9323.02} C_VEL
LIN {X 0,Y 432.336,Z 881.441,A -85,B 0,C 180,E1 -9326.002,E2 -9326.002} C_VEL
LIN {X 0,Y 432.335,Z 881.44,A -85,B 0,C 180,E1 -9329.493,E2 -9329.493} C_VEL
LIN {X 0,Y 432.316,Z 881.442,A -85,B 0,C 180,E1 -9331.871,E2 -9331.871} C_VEL
LIN {X 0,Y 432.319,Z 881.449,A -85,B 0,C 180,E1 -9334.996,E2 -9334.996} C_VEL
LIN {X 0,Y 432.356,Z 881.437,A -85,B 0,C 180,E1 -9338.045,E2 -9338.045} C_VEL
LIN {X 0,Y 432.349,Z 881.443,A -85,B 0,C 180,E1 -9341.027,E2 -9341.027} C_VEL
LIN {X 0,Y 432.365,Z 881.437,A -85,B 0,C 180,E1 -9343.958,E2 -9343.958} C_VEL
LIN {X 0,Y 432.454,Z 881.429,A -85,B 0,C 180,E1 -9347.803,E2 -9347.803} C_VEL
LIN {X 0,Y 432.448,Z 881.432,A -85,B 0,C 180,E1 -9351.589,E2 -9351.589} C_VEL
LIN {X 0,Y 432.552,Z 881.414,A -85,B 0,C 180,E1 -9354.405,E2 -9354.405} C_VEL
LIN {X 0,Y 432.593,Z 881.413,A -85,B 0,C 180,E1 -9358.138,E2 -9358.138} C_VEL
LIN {X 0,Y 432.622,Z 881.411,A -85,B 0,C 180,E1 -9360,E2 -9360} C_VEL
LIN {X 0,Y 432.539,Z 881.415,A -85,B 0,C 180,E1 -9362.794,E2 -9362.794} C_VEL
LIN {X 0,Y 432.551,Z 881.413,A -85,B 0,C 180,E1 -9365.594,E2 -9365.594} C_VEL
LIN {X 0,Y 432.447,Z 881.433,A -85,B 0,C 180,E1 -9368.41,E2 -9368.41} C_VEL
LIN {X 0,Y 432.452,Z 881.427,A -85,B 0,C 180,E1 -9372.196,E2 -9372.196} C_VEL
LIN {X 0,Y 432.363,Z 881.436,A -85,B 0,C 180,E1 -9376.041,E2 -9376.041} C_VEL
LIN {X 0,Y 432.349,Z 881.439,A -85,B 0,C 180,E1 -9379.469,E2 -9379.469} C_VEL
LIN {X 0,Y 432.339,Z 881.439,A -85,B 0,C 180,E1 -9382.092,E2 -9382.092} C_VEL
LIN {X 0,Y 432.312,Z 881.448,A -85,B 0,C 180,E1 -9385.003,E2 -9385.003} C_VEL
LIN {X 0,Y 432.312,Z 881.443,A -85,B 0,C 180,E1 -9388.128,E2 -9388.128} C_VEL
LIN {X 0,Y 432.299,Z 881.45,A -85,B 0,C 180,E1 -9391.347,E2 -9391.347} C_VEL
LIN {X 0,Y 432.321,Z 881.441,A -85,B 0,C 180,E1 -9394.678,E2 -9394.678} C_VEL
LIN {X 0,Y 432.317,Z 881.445,A -85,B 0,C 180,E1 -9398.152,E2 -9398.152} C_VEL
LIN {X 0,Y 432.3,Z 881.45,A -85,B 0,C 180,E1 -9401.801,E2 -9401.801} C_VEL
LIN {X 0,Y 432.331,Z 881.444,A -85,B 0,C 180,E1 -9404.347,E2 -9404.347} C_VEL
LIN {X 0,Y 432.3,Z 881.444,A -85,B 0,C 180,E1 -9407.018,E2 -9407.018} C_VEL
LIN {X 0,Y 432.286,Z 881.448,A -85,B 0,C 180,E1 -9409.828,E2 -9409.828} C_VEL
LIN {X 0,Y 432.292,Z 881.446,A -85,B 0,C 180,E1 -9413.02,E2 -9413.02} C_VEL
LIN {X 0,Y 432.331,Z 881.441,A -85,B 0,C 180,E1 -9416.002,E2 -9416.002} C_VEL
LIN {X 0,Y 432.33,Z 881.44,A -85,B 0,C 180,E1 -9419.493,E2 -9419.493} C_VEL
LIN {X 0,Y 432.311,Z 881.443,A -85,B 0,C 180,E1 -9421.871,E2 -9421.871} C_VEL
LIN {X 0,Y 432.356,Z 881.482,A -85,B 0,C 180,E1 -9424.742,E2 -9424.742} C_VEL
LIN {X 0,Y 434.302,Z 892.256,A -85,B 0,C 180,E1 -9427.278,E2 -9427.278} C_VEL
LIN {X 0,Y 433.59,Z 906.175,A -85,B 0,C 180,E1 -9430.346,E2 -9430.346} C_VEL
LIN {X 0,Y 432.793,Z 921.369,A -85,B 0,C 180,E1 -9433.641,E2 -9433.641} C_VEL
LIN {X 0,Y 432.454,Z 930.286,A -85,B 0,C 180,E1 -9435.56,E2 -9435.56} C_VEL
LIN {X 0,Y 434.852,Z 949.923,A -85,B 0,C 180,E1 -9436.026,E2 -9436.026} C_VEL
LIN {X 0,Y 434.238,Z 1007.719,A -85,B 0,C 180,E1 -9437.112,E2 -9437.112} C_VEL
LIN {X 0,Y 433.908,Z 1017.944,A -85,B 0,C 180,E1 -9437.429,E2 -9437.429} C_VEL
LIN {X 0,Y 433.54,Z 1029.194,A -85,B 0,C 180,E1 -9437.953,E2 -9437.953} C_VEL
LIN {X 0,Y 433.166,Z 1039.754,A -85,B 0,C 180,E1 -9438.654,E2 -9438.654} C_VEL
LIN {X 0,Y 432.797,Z 1048.072,A -85,B 0,C 180,E1 -9439.355,E2 -9439.355} C_VEL
LIN {X 0,Y 432.439,Z 1055.972,A -85,B 0,C 180,E1 -9440.174,E2 -9440.174} C_VEL
LIN {X 0,Y 432.082,Z 1063.37,A -85,B 0,C 180,E1 -9441.111,E2 -9441.111} C_VEL
LIN {X 0,Y 431.752,Z 1070.866,A -85,B 0,C 180,E1 -9442.282,E2 -9442.282} C_VEL
LIN {X 0,Y 431.52,Z 1076.706,A -85,B 0,C 180,E1 -9443.453,E2 -9443.453} C_VEL
LIN {X 0,Y 431.402,Z 1080.54,A -85,B 0,C 180,E1 -9444.39,E2 -9444.39} C_VEL
LIN {X 0,Y 431.268,Z 1084.885,A -85,B 0,C 180,E1 -9445.794,E2 -9445.794} C_VEL
LIN {X 0,Y 431.287,Z 1087.919,A -85,B 0,C 180,E1 -9447.198,E2 -9447.198} C_VEL
LIN {X 0,Y 431.219,Z 1089.241,A -85,B 0,C 180,E1 -9448.132,E2 -9448.132} C_VEL
LIN {X 0,Y 431.19,Z 1090.062,A -85,B 0,C 180,E1 -9449.066,E2 -9449.066} C_VEL
LIN {X 0,Y 431.189,Z 1090.352,A -85,B 0,C 180,E1 -9450,E2 -9450} C_VEL
LIN {X 0,Y 431.19,Z 1090.031,A -85,B 0,C 180,E1 -9450.934,E2 -9450.934} C_VEL
LIN {X 0,Y 431.219,Z 1089.202,A -85,B 0,C 180,E1 -9451.868,E2 -9451.868} C_VEL
LIN {X 0,Y 431.286,Z 1087.87,A -85,B 0,C 180,E1 -9452.802,E2 -9452.802} C_VEL
LIN {X 0,Y 431.267,Z 1084.795,A -85,B 0,C 180,E1 -9454.205,E2 -9454.205} C_VEL
LIN {X 0,Y 431.38,Z 1081.995,A -85,B 0,C 180,E1 -9455.141,E2 -9455.141} C_VEL
LIN {X 0,Y 431.452,Z 1078.054,A -85,B 0,C 180,E1 -9456.194,E2 -9456.194} C_VEL
LIN {X 0,Y 431.651,Z 1073.15,A -85,B 0,C 180,E1 -9457.249,E2 -9457.249} C_VEL
LIN {X 0,Y 431.821,Z 1067.858,A -85,B 0,C 180,E1 -9458.187,E2 -9458.187} C_VEL
LIN {X 0,Y 432.168,Z 1061.492,A -85,B 0,C 180,E1 -9459.123,E2 -9459.123} C_VEL
LIN {X 0,Y 432.501,Z 1054.794,A -85,B 0,C 180,E1 -9459.942,E2 -9459.942} C_VEL
LIN {X 0,Y 432.843,Z 1046.686,A -85,B 0,C 180,E1 -9460.762,E2 -9460.762} C_VEL
LIN {X 0,Y 433.285,Z 1036.583,A -85,B 0,C 180,E1 -9461.579,E2 -9461.579} C_VEL
LIN {X 0,Y 433.656,Z 1025.852,A -85,B 0,C 180,E1 -9462.222,E2 -9462.222} C_VEL
LIN {X 0,Y 433.998,Z 1015.872,A -85,B 0,C 180,E1 -9462.657,E2 -9462.657} C_VEL
LIN {X 0,Y 434.311,Z 1006.18,A -85,B 0,C 180,E1 -9462.945,E2 -9462.945} C_VEL
LIN {X 0,Y 434.823,Z 948.231,A -85,B 0,C 180,E1 -9464.071,E2 -9464.071} C_VEL
LIN {X 0,Y 432.423,Z 929.1,A -85,B 0,C 180,E1 -9464.576,E2 -9464.576} C_VEL
LIN {X 0,Y 433.058,Z 914.618,A -85,B 0,C 180,E1 -9467.715,E2 -9467.715} C_VEL
LIN {X 0,Y 434.006,Z 899.311,A -85,B 0,C 180,E1 -9471.119,E2 -9471.119} C_VEL
LIN {X 0,Y 434.26,Z 892.403,A -85,B 0,C 180,E1 -9472.709,E2 -9472.709} C_VEL
LIN {X 0,Y 432.745,Z 883.336,A -85,B 0,C 180,E1 -9474.977,E2 -9474.977} C_VEL
LIN {X 0,Y 432.352,Z 881.447,A -85,B 0,C 180,E1 -9475.516,E2 -9475.516} C_VEL
LIN {X 0,Y 432.312,Z 881.45,A -85,B 0,C 180,E1 -9479.19,E2 -9479.19} C_VEL
LIN {X 0,Y 432.313,Z 881.447,A -85,B 0,C 180,E1 -9482.444,E2 -9482.444} C_VEL
LIN {X 0,Y 432.329,Z 881.446,A -85,B 0,C 180,E1 -9485.819,E2 -9485.819} C_VEL
LIN {X 0,Y 432.308,Z 881.446,A -85,B 0,C 180,E1 -9488.709,E2 -9488.709} C_VEL
LIN {X 0,Y 432.298,Z 881.45,A -85,B 0,C 180,E1 -9491.801,E2 -9491.801} C_VEL
LIN {X 0,Y 432.329,Z 881.445,A -85,B 0,C 180,E1 -9494.348,E2 -9494.348} C_VEL
LIN {X 0,Y 432.297,Z 881.445,A -85,B 0,C 180,E1 -9497.019,E2 -9497.019} C_VEL
LIN {X 0,Y 432.285,Z 881.452,A -85,B 0,C 180,E1 -9499.828,E2 -9499.828} C_VEL
LIN {X 0,Y 432.291,Z 881.447,A -85,B 0,C 180,E1 -9503.021,E2 -9503.021} C_VEL
LIN {X 0,Y 432.33,Z 881.445,A -85,B 0,C 180,E1 -9506.002,E2 -9506.002} C_VEL
LIN {X 0,Y 432.329,Z 881.443,A -85,B 0,C 180,E1 -9509.494,E2 -9509.494} C_VEL
LIN {X 0,Y 432.31,Z 881.446,A -85,B 0,C 180,E1 -9511.872,E2 -9511.872} C_VEL
LIN {X 0,Y 432.31,Z 881.453,A -85,B 0,C 180,E1 -9514.997,E2 -9514.997} C_VEL
LIN {X 0,Y 432.35,Z 881.445,A -85,B 0,C 180,E1 -9518.046,E2 -9518.046} C_VEL
LIN {X 0,Y 432.375,Z 881.557,A -85,B 0,C 180,E1 -9520.259,E2 -9520.259} C_VEL
LIN {X 0,Y 433.158,Z 887.109,A -85,B 0,C 180,E1 -9522.045,E2 -9522.045} C_VEL
LIN {X 0,Y 432.778,Z 895.162,A -85,B 0,C 180,E1 -9524.458,E2 -9524.458} C_VEL
LIN {X 0,Y 432.634,Z 898.902,A -85,B 0,C 180,E1 -9525.534,E2 -9525.534} C_VEL
LIN {X 0,Y 435.105,Z 912.028,A -85,B 0,C 180,E1 -9525.906,E2 -9525.906} C_VEL
LIN {X 0,Y 434.338,Z 975.811,A -85,B 0,C 180,E1 -9527.175,E2 -9527.175} C_VEL
LIN {X 0,Y 434.051,Z 988.015,A -85,B 0,C 180,E1 -9527.612,E2 -9527.612} C_VEL
LIN {X 0,Y 433.729,Z 996.946,A -85,B 0,C 180,E1 -9528.077,E2 -9528.077} C_VEL
LIN {X 0,Y 433.455,Z 1005.602,A -85,B 0,C 180,E1 -9528.663,E2 -9528.663} C_VEL
LIN {X 0,Y 433.154,Z 1013.901,A -85,B 0,C 180,E1 -9529.365,E2 -9529.365} C_VEL
LIN {X 0,Y 432.758,Z 1021.774,A -85,B 0,C 180,E1 -9530.182,E2 -9530.182} C_VEL
LIN {X 0,Y 432.341,Z 1029.131,A -85,B 0,C 180,E1 -9531.117,E2 -9531.117} C_VEL
LIN {X 0,Y 432.018,Z 1036.565,A -85,B 0,C 180,E1 -9532.287,E2 -9532.287} C_VEL
LIN {X 0,Y 431.875,Z 1042.348,A -85,B 0,C 180,E1 -9533.46,E2 -9533.46} C_VEL
LIN {X 0,Y 431.598,Z 1046.147,A -85,B 0,C 180,E1 -9534.394,E2 -9534.394} C_VEL
LIN {X 0,Y 431.41,Z 1049.215,A -85,B 0,C 180,E1 -9535.328,E2 -9535.328} C_VEL
LIN {X 0,Y 431.464,Z 1051.595,A -85,B 0,C 180,E1 -9536.265,E2 -9536.265} C_VEL
LIN {X 0,Y 431.332,Z 1053.422,A -85,B 0,C 180,E1 -9537.199,E2 -9537.199} C_VEL
LIN {X 0,Y 431.249,Z 1054.728,A -85,B 0,C 180,E1 -9538.133,E2 -9538.133} C_VEL
LIN {X 0,Y 431.194,Z 1055.536,A -85,B 0,C 180,E1 -9539.067,E2 -9539.067} C_VEL
LIN {X 0,Y 431.191,Z 1055.82,A -85,B 0,C 180,E1 -9540,E2 -9540} C_VEL
LIN {X 0,Y 431.193,Z 1055.501,A -85,B 0,C 180,E1 -9540.934,E2 -9540.934} C_VEL
LIN {X 0,Y 431.239,Z 1054.681,A -85,B 0,C 180,E1 -9541.868,E2 -9541.868} C_VEL
LIN {X 0,Y 431.325,Z 1053.363,A -85,B 0,C 180,E1 -9542.802,E2 -9542.802} C_VEL
LIN {X 0,Y 431.412,Z 1050.338,A -85,B 0,C 180,E1 -9544.204,E2 -9544.204} C_VEL
LIN {X 0,Y 431.45,Z 1047.575,A -85,B 0,C 180,E1 -9545.141,E2 -9545.141} C_VEL
LIN {X 0,Y 431.705,Z 1044.165,A -85,B 0,C 180,E1 -9546.075,E2 -9546.075} C_VEL
LIN {X 0,Y 431.828,Z 1039.237,A -85,B 0,C 180,E1 -9547.167,E2 -9547.167} C_VEL
LIN {X 0,Y 432.069,Z 1033.591,A -85,B 0,C 180,E1 -9548.183,E2 -9548.183} C_VEL
LIN {X 0,Y 432.366,Z 1027.271,A -85,B 0,C 180,E1 -9549.119,E2 -9549.119} C_VEL
LIN {X 0,Y 432.735,Z 1019.588,A -85,B 0,C 180,E1 -9550.055,E2 -9550.055} C_VEL
LIN {X 0,Y 433.194,Z 1010.048,A -85,B 0,C 180,E1 -9550.99,E2 -9550.99} C_VEL
LIN {X 0,Y 433.572,Z 1000.733,A -85,B 0,C 180,E1 -9551.691,E2 -9551.691} C_VEL
LIN {X 0,Y 433.799,Z 991.785,A -85,B 0,C 180,E1 -9552.218,E2 -9552.218} C_VEL
LIN {X 0,Y 434.032,Z 981.755,A -85,B 0,C 180,E1 -9552.657,E2 -9552.657} C_VEL
LIN {X 0,Y 434.281,Z 971.887,A -85,B 0,C 180,E1 -9552.947,E2 -9552.947} C_VEL
LIN {X 0,Y 434.835,Z 911.714,A -85,B 0,C 180,E1 -9554.073,E2 -9554.073} C_VEL
LIN {X 0,Y 432.361,Z 897.286,A -85,B 0,C 180,E1 -9554.451,E2 -9554.451} C_VEL
LIN {X 0,Y 432.774,Z 886.448,A -85,B 0,C 180,E1 -9557.484,E2 -9557.484} C_VEL
LIN {X 0,Y 432.417,Z 881.437,A -85,B 0,C 180,E1 -9558.97,E2 -9558.97} C_VEL
LIN {X 0,Y 432.34,Z 881.439,A -85,B 0,C 180,E1 -9562.093,E2 -9562.093} C_VEL
LIN {X 0,Y 432.313,Z 881.447,A -85,B 0,C 180,E1 -9565.004,E2 -9565.004} C_VEL
LIN {X 0,Y 432.313,Z 881.443,A -85,B 0,C 180,E1 -9568.129,E2 -9568.129} C_VEL
LIN {X 0,Y 432.305,Z 881.449,A -85,B 0,C 180,E1 -9571.348,E2 -9571.348} C_VEL
LIN {X 0,Y 432.327,Z 881.441,A -85,B 0,C 180,E1 -9574.679,E2 -9574.679} C_VEL
LIN {X 0,Y 432.32,Z 881.444,A -85,B 0,C 180,E1 -9578.152,E2 -9578.152} C_VEL
LIN {X 0,Y 432.302,Z 881.449,A -85,B 0,C 180,E1 -9581.802,E2 -9581.802} C_VEL
LIN {X 0,Y 432.334,Z 881.444,A -85,B 0,C 180,E1 -9584.348,E2 -9584.348} C_VEL
LIN {X 0,Y 432.303,Z 881.444,A -85,B 0,C 180,E1 -9587.019,E2 -9587.019} C_VEL
LIN {X 0,Y 432.289,Z 881.447,A -85,B 0,C 180,E1 -9589.829,E2 -9589.829} C_VEL
LIN {X 0,Y 432.297,Z 881.446,A -85,B 0,C 180,E1 -9593.021,E2 -9593.021} C_VEL
LIN {X 0,Y 432.335,Z 881.441,A -85,B 0,C 180,E1 -9596.003,E2 -9596.003} C_VEL
LIN {X 0,Y 432.334,Z 881.44,A -85,B 0,C 180,E1 -9599.494,E2 -9599.494} C_VEL
LIN {X 0,Y 432.315,Z 881.442,A -85,B 0,C 180,E1 -9601.872,E2 -9601.872} C_VEL
LIN {X 0,Y 432.319,Z 881.449,A -85,B 0,C 180,E1 -9604.997,E2 -9604.997} C_VEL
LIN {X 0,Y 432.356,Z 881.437,A -85,B 0,C 180,E1 -9608.046,E2 -9608.046} C_VEL
LIN {X 0,Y 432.349,Z 881.443,A -85,B 0,C 180,E1 -9611.028,E2 -9611.028} C_VEL
LIN {X 0,Y 432.425,Z 881.43,A -85,B 0,C 180,E1 -9613.961,E2 -9613.961} C_VEL
LIN {X 0,Y 432.455,Z 881.429,A -85,B 0,C 180,E1 -9617.803,E2 -9617.803} C_VEL
LIN {X 0,Y 432.45,Z 881.431,A -85,B 0,C 180,E1 -9621.59,E2 -9621.59} C_VEL
LIN {X 0,Y 432.554,Z 881.414,A -85,B 0,C 180,E1 -9624.406,E2 -9624.406} C_VEL
LIN {X 0,Y 431.779,Z 881.51,A -85,B 0,C 180,E1 -9625.183,E2 -9625.183} C_VEL
LIN {X 0,Y 428.972,Z 881.861,A -85,B 0,C 180,E1 -9626.446,E2 -9626.446} C_VEL
LIN {X 0,Y 426.642,Z 882.154,A -85,B 0,C 180,E1 -9627.466,E2 -9627.466} C_VEL
LIN {X 0,Y 425.605,Z 882.283,A -85,B 0,C 180,E1 -9628.253,E2 -9628.253} C_VEL
LIN {X 0,Y 425.495,Z 882.293,A -85,B 0,C 180,E1 -9628.519,E2 -9628.519} C_VEL
LIN {X 0,Y 425.576,Z 882.288,A -85,B 0,C 180,E1 -9630,E2 -9630} C_VEL
LIN {X 0,Y 425.498,Z 882.292,A -85,B 0,C 180,E1 -9632.84,E2 -9632.84} C_VEL
LIN {X 0,Y 425.512,Z 882.29,A -85,B 0,C 180,E1 -9635.688,E2 -9635.688} C_VEL
LIN {X 0,Y 425.398,Z 882.31,A -85,B 0,C 180,E1 -9638.551,E2 -9638.551} C_VEL
LIN {X 0,Y 425.411,Z 882.307,A -85,B 0,C 180,E1 -9642.402,E2 -9642.402} C_VEL
LIN {X 0,Y 425.318,Z 882.316,A -85,B 0,C 180,E1 -9646.315,E2 -9646.315} C_VEL
LIN {X 0,Y 425.302,Z 882.317,A -85,B 0,C 180,E1 -9649.623,E2 -9649.623} C_VEL
LIN {X 0,Y 425.289,Z 882.318,A -85,B 0,C 180,E1 -9652.339,E2 -9652.339} C_VEL
LIN {X 0,Y 425.253,Z 882.326,A -85,B 0,C 180,E1 -9655.448,E2 -9655.448} C_VEL
LIN {X 0,Y 425.3,Z 882.318,A -85,B 0,C 180,E1 -9658.857,E2 -9658.857} C_VEL
LIN {X 0,Y 425.25,Z 882.325,A -85,B 0,C 180,E1 -9661.929,E2 -9661.929} C_VEL
LIN {X 0,Y 425.293,Z 882.32,A -85,B 0,C 180,E1 -9665.337,E2 -9665.337} C_VEL
LIN {X 0,Y 425.276,Z 882.319,A -85,B 0,C 180,E1 -9668.901,E2 -9668.901} C_VEL
LIN {X 0,Y 425.258,Z 882.322,A -85,B 0,C 180,E1 -9672.656,E2 -9672.656} C_VEL
LIN {X 0,Y 425.287,Z 882.318,A -85,B 0,C 180,E1 -9675.283,E2 -9675.283} C_VEL
LIN {X 0,Y 425.248,Z 882.325,A -85,B 0,C 180,E1 -9678.617,E2 -9678.617} C_VEL
LIN {X 0,Y 425.271,Z 882.326,A -85,B 0,C 180,E1 -9682.304,E2 -9682.304} C_VEL
LIN {X 0,Y 425.289,Z 882.318,A -85,B 0,C 180,E1 -9685.815,E2 -9685.815} C_VEL
LIN {X 0,Y 425.289,Z 882.319,A -85,B 0,C 180,E1 -9689.24,E2 -9689.24} C_VEL
LIN {X 0,Y 425.241,Z 882.326,A -85,B 0,C 180,E1 -9692.434,E2 -9692.434} C_VEL
LIN {X 0,Y 425.319,Z 882.315,A -85,B 0,C 180,E1 -9695.6,E2 -9695.6} C_VEL
LIN {X 0,Y 425.286,Z 882.32,A -85,B 0,C 180,E1 -9698.681,E2 -9698.681} C_VEL
LIN {X 0,Y 425.299,Z 882.318,A -85,B 0,C 180,E1 -9701.701,E2 -9701.701} C_VEL
LIN {X 0,Y 425.286,Z 882.318,A -85,B 0,C 180,E1 -9704.668,E2 -9704.668} C_VEL
LIN {X 0,Y 425.41,Z 882.309,A -85,B 0,C 180,E1 -9707.598,E2 -9707.598} C_VEL
LIN {X 0,Y 425.396,Z 882.308,A -85,B 0,C 180,E1 -9711.449,E2 -9711.449} C_VEL
LIN {X 0,Y 425.51,Z 882.292,A -85,B 0,C 180,E1 -9714.312,E2 -9714.312} C_VEL
LIN {X 0,Y 425.562,Z 882.289,A -85,B 0,C 180,E1 -9718.107,E2 -9718.107} C_VEL
LIN {X 0,Y 425.574,Z 882.289,A -85,B 0,C 180,E1 -9720,E2 -9720} C_VEL
LIN {X 0,Y 425.496,Z 882.292,A -85,B 0,C 180,E1 -9722.84,E2 -9722.84} C_VEL
LIN {X 0,Y 425.51,Z 882.291,A -85,B 0,C 180,E1 -9725.687,E2 -9725.687} C_VEL
LIN {X 0,Y 425.395,Z 882.31,A -85,B 0,C 180,E1 -9728.551,E2 -9728.551} C_VEL
LIN {X 0,Y 425.408,Z 882.307,A -85,B 0,C 180,E1 -9732.402,E2 -9732.402} C_VEL
LIN {X 0,Y 425.315,Z 882.316,A -85,B 0,C 180,E1 -9736.314,E2 -9736.314} C_VEL
LIN {X 0,Y 425.298,Z 882.317,A -85,B 0,C 180,E1 -9739.623,E2 -9739.623} C_VEL
LIN {X 0,Y 425.285,Z 882.318,A -85,B 0,C 180,E1 -9742.338,E2 -9742.338} C_VEL
LIN {X 0,Y 425.249,Z 882.326,A -85,B 0,C 180,E1 -9745.448,E2 -9745.448} C_VEL
LIN {X 0,Y 425.296,Z 882.318,A -85,B 0,C 180,E1 -9748.857,E2 -9748.857} C_VEL
LIN {X 0,Y 425.245,Z 882.325,A -85,B 0,C 180,E1 -9751.928,E2 -9751.928} C_VEL
LIN {X 0,Y 425.289,Z 882.321,A -85,B 0,C 180,E1 -9755.337,E2 -9755.337} C_VEL
LIN {X 0,Y 425.272,Z 882.319,A -85,B 0,C 180,E1 -9758.901,E2 -9758.901} C_VEL
LIN {X 0,Y 425.253,Z 882.322,A -85,B 0,C 180,E1 -9762.655,E2 -9762.655} C_VEL
LIN {X 0,Y 425.283,Z 882.318,A -85,B 0,C 180,E1 -9765.283,E2 -9765.283} C_VEL
LIN {X 0,Y 425.244,Z 882.326,A -85,B 0,C 180,E1 -9768.617,E2 -9768.617} C_VEL
LIN {X 0,Y 425.266,Z 882.327,A -85,B 0,C 180,E1 -9772.304,E2 -9772.304} C_VEL
LIN {X 0,Y 425.284,Z 882.318,A -85,B 0,C 180,E1 -9775.815,E2 -9775.815} C_VEL
LIN {X 0,Y 425.284,Z 882.319,A -85,B 0,C 180,E1 -9779.24,E2 -9779.24} C_VEL
LIN {X 0,Y 425.236,Z 882.327,A -85,B 0,C 180,E1 -9782.434,E2 -9782.434} C_VEL
LIN {X 0,Y 425.357,Z 882.505,A -85,B 0,C 180,E1 -9784.609,E2 -9784.609} C_VEL
LIN {X 0,Y 427.242,Z 892.89,A -85,B 0,C 180,E1 -9787.099,E2 -9787.099} C_VEL
LIN {X 0,Y 426.709,Z 905.144,A -85,B 0,C 180,E1 -9789.851,E2 -9789.851} C_VEL
LIN {X 0,Y 425.828,Z 920.842,A -85,B 0,C 180,E1 -9793.319,E2 -9793.319} C_VEL
LIN {X 0,Y 425.402,Z 930.104,A -85,B 0,C 180,E1 -9795.346,E2 -9795.346} C_VEL
LIN {X 0,Y 427.925,Z 950.19,A -85,B 0,C 180,E1 -9795.824,E2 -9795.824} C_VEL
LIN {X 0,Y 427.27,Z 1008.437,A -85,B 0,C 180,E1 -9796.958,E2 -9796.958} C_VEL
LIN {X 0,Y 426.869,Z 1019.845,A -85,B 0,C 180,E1 -9797.339,E2 -9797.339} C_VEL
LIN {X 0,Y 426.509,Z 1030.231,A -85,B 0,C 180,E1 -9797.872,E2 -9797.872} C_VEL
LIN {X 0,Y 426.186,Z 1039.016,A -85,B 0,C 180,E1 -9798.466,E2 -9798.466} C_VEL
LIN {X 0,Y 425.805,Z 1047.423,A -85,B 0,C 180,E1 -9799.178,E2 -9799.178} C_VEL
LIN {X 0,Y 425.394,Z 1055.391,A -85,B 0,C 180,E1 -9800.01,E2 -9800.01} C_VEL
LIN {X 0,Y 425.039,Z 1062.851,A -85,B 0,C 180,E1 -9800.962,E2 -9800.962} C_VEL
LIN {X 0,Y 424.688,Z 1070.413,A -85,B 0,C 180,E1 -9802.153,E2 -9802.153} C_VEL
LIN {X 0,Y 424.441,Z 1076.784,A -85,B 0,C 180,E1 -9803.459,E2 -9803.459} C_VEL
LIN {X 0,Y 424.311,Z 1080.167,A -85,B 0,C 180,E1 -9804.296,E2 -9804.296} C_VEL
LIN {X 0,Y 424.189,Z 1084.547,A -85,B 0,C 180,E1 -9805.724,E2 -9805.724} C_VEL
LIN {X 0,Y 424.186,Z 1087.599,A -85,B 0,C 180,E1 -9807.151,E2 -9807.151} C_VEL
LIN {X 0,Y 424.146,Z 1088.938,A -85,B 0,C 180,E1 -9808.101,E2 -9808.101} C_VEL
LIN {X 0,Y 424.108,Z 1089.77,A -85,B 0,C 180,E1 -9809.05,E2 -9809.05} C_VEL
LIN {X 0,Y 424.105,Z 1090.063,A -85,B 0,C 180,E1 -9810,E2 -9810} C_VEL
LIN {X 0,Y 424.108,Z 1089.747,A -85,B 0,C 180,E1 -9810.949,E2 -9810.949} C_VEL
LIN {X 0,Y 424.145,Z 1088.926,A -85,B 0,C 180,E1 -9811.899,E2 -9811.899} C_VEL
LIN {X 0,Y 424.184,Z 1087.598,A -85,B 0,C 180,E1 -9812.849,E2 -9812.849} C_VEL
LIN {X 0,Y 424.189,Z 1084.534,A -85,B 0,C 180,E1 -9814.276,E2 -9814.276} C_VEL
LIN {X 0,Y 424.296,Z 1081.737,A -85,B 0,C 180,E1 -9815.227,E2 -9815.227} C_VEL
LIN {X 0,Y 424.458,Z 1076.29,A -85,B 0,C 180,E1 -9816.656,E2 -9816.656} C_VEL
LIN {X 0,Y 424.724,Z 1069.042,A -85,B 0,C 180,E1 -9818.085,E2 -9818.085} C_VEL
LIN {X 0,Y 425.038,Z 1062.951,A -85,B 0,C 180,E1 -9819.037,E2 -9819.037} C_VEL
LIN {X 0,Y 425.448,Z 1055.541,A -85,B 0,C 180,E1 -9819.988,E2 -9819.988} C_VEL
LIN {X 0,Y 425.784,Z 1047.63,A -85,B 0,C 180,E1 -9820.822,E2 -9820.822} C_VEL
LIN {X 0,Y 426.189,Z 1039.33,A -85,B 0,C 180,E1 -9821.534,E2 -9821.534} C_VEL
LIN {X 0,Y 426.587,Z 1028.888,A -85,B 0,C 180,E1 -9822.246,E2 -9822.246} C_VEL
LIN {X 0,Y 427.017,Z 1017.357,A -85,B 0,C 180,E1 -9822.807,E2 -9822.807} C_VEL
LIN {X 0,Y 427.361,Z 1007.492,A -85,B 0,C 180,E1 -9823.129,E2 -9823.129} C_VEL
LIN {X 0,Y 427.958,Z 948.516,A -85,B 0,C 180,E1 -9824.326,E2 -9824.326} C_VEL
LIN {X 0,Y 425.413,Z 928.809,A -85,B 0,C 180,E1 -9824.855,E2 -9824.855} C_VEL
LIN {X 0,Y 426.102,Z 914.573,A -85,B 0,C 180,E1 -9828.014,E2 -9828.014} C_VEL
LIN {X 0,Y 427.075,Z 899.375,A -85,B 0,C 180,E1 -9831.478,E2 -9831.478} C_VEL
LIN {X 0,Y 427.283,Z 893.297,A -85,B 0,C 180,E1 -9832.914,E2 -9832.914} C_VEL
LIN {X 0,Y 425.584,Z 883.613,A -85,B 0,C 180,E1 -9835.427,E2 -9835.427} C_VEL
LIN {X 0,Y 425.277,Z 882.328,A -85,B 0,C 180,E1 -9835.84,E2 -9835.84} C_VEL
LIN {X 0,Y 425.293,Z 882.324,A -85,B 0,C 180,E1 -9838.857,E2 -9838.857} C_VEL
LIN {X 0,Y 425.25,Z 882.328,A -85,B 0,C 180,E1 -9841.928,E2 -9841.928} C_VEL
LIN {X 0,Y 425.289,Z 882.324,A -85,B 0,C 180,E1 -9845.337,E2 -9845.337} C_VEL
LIN {X 0,Y 425.261,Z 882.324,A -85,B 0,C 180,E1 -9848.903,E2 -9848.903} C_VEL
LIN {X 0,Y 425.26,Z 882.326,A -85,B 0,C 180,E1 -9851.954,E2 -9851.954} C_VEL
LIN {X 0,Y 425.281,Z 882.322,A -85,B 0,C 180,E1 -9855.284,E2 -9855.284} C_VEL
LIN {X 0,Y 425.242,Z 882.326,A -85,B 0,C 180,E1 -9858.618,E2 -9858.618} C_VEL
LIN {X 0,Y 425.265,Z 882.326,A -85,B 0,C 180,E1 -9862.305,E2 -9862.305} C_VEL
LIN {X 0,Y 425.283,Z 882.321,A -85,B 0,C 180,E1 -9865.815,E2 -9865.815} C_VEL
LIN {X 0,Y 425.283,Z 882.321,A -85,B 0,C 180,E1 -9869.241,E2 -9869.241} C_VEL
LIN {X 0,Y 425.236,Z 882.331,A -85,B 0,C 180,E1 -9872.435,E2 -9872.435} C_VEL
LIN {X 0,Y 425.31,Z 882.323,A -85,B 0,C 180,E1 -9875.6,E2 -9875.6} C_VEL
LIN {X 0,Y 425.281,Z 882.328,A -85,B 0,C 180,E1 -9878.681,E2 -9878.681} C_VEL
LIN {X 0,Y 425.305,Z 882.401,A -85,B 0,C 180,E1 -9879.979,E2 -9879.979} C_VEL
LIN {X 0,Y 426.165,Z 887.725,A -85,B 0,C 180,E1 -9881.74,E2 -9881.74} C_VEL
LIN {X 0,Y 425.964,Z 894.118,A -85,B 0,C 180,E1 -9883.711,E2 -9883.711} C_VEL
LIN {X 0,Y 425.67,Z 899.222,A -85,B 0,C 180,E1 -9885.243,E2 -9885.243} C_VEL
LIN {X 0,Y 428.352,Z 913.145,A -85,B 0,C 180,E1 -9885.66,E2 -9885.66} C_VEL
LIN {X 0,Y 427.473,Z 975.665,A -85,B 0,C 180,E1 -9886.935,E2 -9886.935} C_VEL
LIN {X 0,Y 427.188,Z 987.428,A -85,B 0,C 180,E1 -9887.349,E2 -9887.349} C_VEL
LIN {X 0,Y 426.803,Z 997.451,A -85,B 0,C 180,E1 -9887.881,E2 -9887.881} C_VEL
LIN {X 0,Y 426.524,Z 1006.035,A -85,B 0,C 180,E1 -9888.476,E2 -9888.476} C_VEL
LIN {X 0,Y 426.199,Z 1014.287,A -85,B 0,C 180,E1 -9889.189,E2 -9889.189} C_VEL
LIN {X 0,Y 425.792,Z 1022.127,A -85,B 0,C 180,E1 -9890.02,E2 -9890.02} C_VEL
LIN {X 0,Y 425.352,Z 1029.475,A -85,B 0,C 180,E1 -9890.97,E2 -9890.97} C_VEL
